LIN {X 0,Y 460.459,Z 388.647,A -85,B 0,C 180,E1 -8093.427,E2 -8093.427} C_VEL
LIN {X 0,Y 460.171,Z 393.017,A -85,B 0,C 180,E1 -8094.742,E2 -8094.742} C_VEL
LIN {X 0,Y 460.177,Z 395.283,A -85,B 0,C 180,E1 -8095.621,E2 -8095.621} C_VEL
LIN {X 0,Y 459.997,Z 397.136,A -85,B 0,C 180,E1 -8096.496,E2 -8096.496} C_VEL
LIN {X 0,Y 459.827,Z 398.543,A -85,B 0,C 180,E1 -8097.372,E2 -8097.372} C_VEL
LIN {X 0,Y 459.708,Z 400.055,A -85,B 0,C 180,E1 -8099.124,E2 -8099.124} C_VEL
LIN {X 0,Y 459.693,Z 400.219,A -85,B 0,C 180,E1 -8100,E2 -8100} C_VEL
LIN {X 0,Y 459.693,Z 399.948,A -85,B 0,C 180,E1 -8100.876,E2 -8100.876} C_VEL
LIN {X 0,Y 459.808,Z 398.188,A -85,B 0,C 180,E1 -8102.628,E2 -8102.628} C_VEL
LIN {X 0,Y 459.991,Z 396.689,A -85,B 0,C 180,E1 -8103.504,E2 -8103.504} C_VEL
LIN {X 0,Y 460.089,Z 393.615,A -85,B 0,C 180,E1 -8104.819,E2 -8104.819} C_VEL
LIN {X 0,Y 460.187,Z 388.427,A -85,B 0,C 180,E1 -8106.417,E2 -8106.417} C_VEL
LIN {X 0,Y 460.472,Z 382.079,A -85,B 0,C 180,E1 -8107.895,E2 -8107.895} C_VEL
LIN {X 0,Y 460.797,Z 374.875,A -85,B 0,C 180,E1 -8109.215,E2 -8109.215} C_VEL
LIN {X 0,Y 461.181,Z 365.885,A -85,B 0,C 180,E1 -8110.537,E2 -8110.537} C_VEL
LIN {X 0,Y 461.678,Z 356.667,A -85,B 0,C 180,E1 -8111.637,E2 -8111.637} C_VEL
LIN {X 0,Y 462.105,Z 346.45,A -85,B 0,C 180,E1 -8112.628,E2 -8112.628} C_VEL
LIN {X 0,Y 462.457,Z 334.22,A -85,B 0,C 180,E1 -8113.58,E2 -8113.58} C_VEL
LIN {X 0,Y 462.892,Z 322.561,A -85,B 0,C 180,E1 -8114.284,E2 -8114.284} C_VEL
LIN {X 0,Y 463.049,Z 309.71,A -85,B 0,C 180,E1 -8114.868,E2 -8114.868} C_VEL
LIN {X 0,Y 459.93,Z 296.427,A -85,B 0,C 180,E1 -8115.404,E2 -8115.404} C_VEL
LIN {X 0,Y 459.882,Z 292.523,A -85,B 0,C 180,E1 -8118.719,E2 -8118.719} C_VEL
LIN {X 0,Y 460.011,Z 292.186,A -85,B 0,C 180,E1 -8120.573,E2 -8120.573} C_VEL
LIN {X 0,Y 460.393,Z 292.14,A -85,B 0,C 180,E1 -8123.664,E2 -8123.664} C_VEL
LIN {X 0,Y 460.54,Z 292.115,A -85,B 0,C 180,E1 -8126.267,E2 -8126.267} C_VEL
LIN {X 0,Y 460.542,Z 292.115,A -85,B 0,C 180,E1 -8129.231,E2 -8129.231} C_VEL
LIN {X 0,Y 460.534,Z 292.118,A -85,B 0,C 180,E1 -8132.284,E2 -8132.284} C_VEL
LIN {X 0,Y 460.513,Z 292.115,A -85,B 0,C 180,E1 -8135.446,E2 -8135.446} C_VEL
LIN {X 0,Y 460.547,Z 292.114,A -85,B 0,C 180,E1 -8138.898,E2 -8138.898} C_VEL
LIN {X 0,Y 460.526,Z 292.123,A -85,B 0,C 180,E1 -8142.181,E2 -8142.181} C_VEL
LIN {X 0,Y 460.52,Z 292.119,A -85,B 0,C 180,E1 -8145.412,E2 -8145.412} C_VEL
LIN {X 0,Y 460.535,Z 292.117,A -85,B 0,C 180,E1 -8148.398,E2 -8148.398} C_VEL
LIN {X 0,Y 460.529,Z 292.12,A -85,B 0,C 180,E1 -8151.267,E2 -8151.267} C_VEL
LIN {X 0,Y 460.47,Z 292.127,A -85,B 0,C 180,E1 -8154.551,E2 -8154.551} C_VEL
LIN {X 0,Y 460.258,Z 292.271,A -85,B 0,C 180,E1 -8156.723,E2 -8156.723} C_VEL
LIN {X 0,Y 460.072,Z 297.348,A -85,B 0,C 180,E1 -8159.728,E2 -8159.728} C_VEL
LIN {X 0,Y 460.018,Z 302.263,A -85,B 0,C 180,E1 -8162.72,E2 -8162.72} C_VEL
LIN {X 0,Y 459.986,Z 307.025,A -85,B 0,C 180,E1 -8165.636,E2 -8165.636} C_VEL
LIN {X 0,Y 459.934,Z 312.249,A -85,B 0,C 180,E1 -8168.767,E2 -8168.767} C_VEL
LIN {X 0,Y 459.91,Z 316.705,A -85,B 0,C 180,E1 -8171.342,E2 -8171.342} C_VEL
LIN {X 0,Y 459.853,Z 320.715,A -85,B 0,C 180,E1 -8173.53,E2 -8173.53} C_VEL
LIN {X 0,Y 459.768,Z 322.003,A -85,B 0,C 180,E1 -8173.864,E2 -8173.864} C_VEL
LIN {X 0,Y 459.446,Z 324.926,A -85,B 0,C 180,E1 -8174.21,E2 -8174.21} C_VEL
LIN {X 0,Y 458.82,Z 329.649,A -85,B 0,C 180,E1 -8174.511,E2 -8174.511} C_VEL
LIN {X 0,Y 458.222,Z 333.723,A -85,B 0,C 180,E1 -8174.684,E2 -8174.684} C_VEL
LIN {X 0,Y 456.634,Z 345.505,A -85,B 0,C 180,E1 -8175.091,E2 -8175.091} C_VEL
LIN {X 0,Y 456.445,Z 349.068,A -85,B 0,C 180,E1 -8175.266,E2 -8175.266} C_VEL
LIN {X 0,Y 455.948,Z 360.679,A -85,B 0,C 180,E1 -8175.94,E2 -8175.94} C_VEL
LIN {X 0,Y 455.497,Z 371.287,A -85,B 0,C 180,E1 -8176.732,E2 -8176.732} C_VEL
LIN {X 0,Y 454.998,Z 382.032,A -85,B 0,C 180,E1 -8177.738,E2 -8177.738} C_VEL
LIN {X 0,Y 454.451,Z 391.614,A -85,B 0,C 180,E1 -8178.854,E2 -8178.854} C_VEL
LIN {X 0,Y 453.896,Z 400.92,A -85,B 0,C 180,E1 -8180.193,E2 -8180.193} C_VEL
LIN {X 0,Y 453.463,Z 408.307,A -85,B 0,C 180,E1 -8181.533,E2 -8181.533} C_VEL
LIN {X 0,Y 453.083,Z 415.107,A -85,B 0,C 180,E1 -8183.093,E2 -8183.093} C_VEL
LIN {X 0,Y 452.857,Z 418.931,A -85,B 0,C 180,E1 -8184.21,E2 -8184.21} C_VEL
LIN {X 0,Y 452.825,Z 422.513,A -85,B 0,C 180,E1 -8185.549,E2 -8185.549} C_VEL
LIN {X 0,Y 452.731,Z 424.363,A -85,B 0,C 180,E1 -8186.44,E2 -8186.44} C_VEL
LIN {X 0,Y 452.673,Z 425.775,A -85,B 0,C 180,E1 -8187.33,E2 -8187.33} C_VEL
LIN {X 0,Y 452.496,Z 427.385,A -85,B 0,C 180,E1 -8189.11,E2 -8189.11} C_VEL
LIN {X 0,Y 452.477,Z 427.621,A -85,B 0,C 180,E1 -8190,E2 -8190} C_VEL
LIN {X 0,Y 452.581,Z 426.849,A -85,B 0,C 180,E1 -8191.78,E2 -8191.78} C_VEL
LIN {X 0,Y 452.673,Z 425.886,A -85,B 0,C 180,E1 -8192.67,E2 -8192.67} C_VEL
LIN {X 0,Y 452.729,Z 424.535,A -85,B 0,C 180,E1 -8193.56,E2 -8193.56} C_VEL
LIN {X 0,Y 452.765,Z 421.693,A -85,B 0,C 180,E1 -8194.898,E2 -8194.898} C_VEL
LIN {X 0,Y 453.005,Z 417.822,A -85,B 0,C 180,E1 -8196.235,E2 -8196.235} C_VEL
LIN {X 0,Y 453.212,Z 412.816,A -85,B 0,C 180,E1 -8197.574,E2 -8197.574} C_VEL
LIN {X 0,Y 453.552,Z 406.493,A -85,B 0,C 180,E1 -8198.914,E2 -8198.914} C_VEL
LIN {X 0,Y 453.999,Z 398.632,A -85,B 0,C 180,E1 -8200.255,E2 -8200.255} C_VEL
LIN {X 0,Y 454.539,Z 390.597,A -85,B 0,C 180,E1 -8201.37,E2 -8201.37} C_VEL
LIN {X 0,Y 455.041,Z 380.753,A -85,B 0,C 180,E1 -8202.488,E2 -8202.488} C_VEL
LIN {X 0,Y 455.56,Z 369.521,A -85,B 0,C 180,E1 -8203.505,E2 -8203.505} C_VEL
LIN {X 0,Y 456.064,Z 358.809,A -85,B 0,C 180,E1 -8204.274,E2 -8204.274} C_VEL
LIN {X 0,Y 456.506,Z 346.692,A -85,B 0,C 180,E1 -8204.944,E2 -8204.944} C_VEL
LIN {X 0,Y 456.499,Z 339.201,A -85,B 0,C 180,E1 -8205.272,E2 -8205.272} C_VEL
LIN {X 0,Y 453.913,Z 327.065,A -85,B 0,C 180,E1 -8205.763,E2 -8205.763} C_VEL
LIN {X 0,Y 452.874,Z 322.749,A -85,B 0,C 180,E1 -8205.923,E2 -8205.923} C_VEL
LIN {X 0,Y 452.824,Z 317.039,A -85,B 0,C 180,E1 -8209.022,E2 -8209.022} C_VEL
LIN {X 0,Y 452.888,Z 312.118,A -85,B 0,C 180,E1 -8211.866,E2 -8211.866} C_VEL
LIN {X 0,Y 452.934,Z 307.318,A -85,B 0,C 180,E1 -8214.768,E2 -8214.768} C_VEL
LIN {X 0,Y 452.967,Z 302.337,A -85,B 0,C 180,E1 -8217.824,E2 -8217.824} C_VEL
LIN {X 0,Y 453.025,Z 297.475,A -85,B 0,C 180,E1 -8220.794,E2 -8220.794} C_VEL
LIN {X 0,Y 453.233,Z 293.034,A -85,B 0,C 180,E1 -8223.49,E2 -8223.49} C_VEL
LIN {X 0,Y 453.443,Z 293.004,A -85,B 0,C 180,E1 -8226.297,E2 -8226.297} C_VEL
LIN {X 0,Y 453.492,Z 292.998,A -85,B 0,C 180,E1 -8229.45,E2 -8229.45} C_VEL
LIN {X 0,Y 453.479,Z 292.999,A -85,B 0,C 180,E1 -8231.935,E2 -8231.935} C_VEL
LIN {X 0,Y 453.486,Z 292.998,A -85,B 0,C 180,E1 -8235.471,E2 -8235.471} C_VEL
LIN {X 0,Y 453.482,Z 292.997,A -85,B 0,C 180,E1 -8238.209,E2 -8238.209} C_VEL
LIN {X 0,Y 453.518,Z 292.993,A -85,B 0,C 180,E1 -8240.79,E2 -8240.79} C_VEL
LIN {X 0,Y 453.42,Z 293.008,A -85,B 0,C 180,E1 -8243.914,E2 -8243.914} C_VEL
LIN {X 0,Y 453.295,Z 293.022,A -85,B 0,C 180,E1 -8246.072,E2 -8246.072} C_VEL
LIN {X 0,Y 453.177,Z 293.167,A -85,B 0,C 180,E1 -8246.951,E2 -8246.951} C_VEL
LIN {X 0,Y 453.012,Z 298.953,A -85,B 0,C 180,E1 -8250.318,E2 -8250.318} C_VEL
LIN {X 0,Y 452.951,Z 303.959,A -85,B 0,C 180,E1 -8253.258,E2 -8253.258} C_VEL
LIN {X 0,Y 452.915,Z 309.103,A -85,B 0,C 180,E1 -8256.28,E2 -8256.28} C_VEL
LIN {X 0,Y 452.914,Z 313.849,A -85,B 0,C 180,E1 -8259.09,E2 -8259.09} C_VEL
LIN {X 0,Y 452.832,Z 318.65,A -85,B 0,C 180,E1 -8261.916,E2 -8261.916} C_VEL
LIN {X 0,Y 452.875,Z 323.053,A -85,B 0,C 180,E1 -8264.475,E2 -8264.475} C_VEL
LIN {X 0,Y 455.889,Z 337.844,A -85,B 0,C 180,E1 -8265.05,E2 -8265.05} C_VEL
LIN {X 0,Y 455.849,Z 347.577,A -85,B 0,C 180,E1 -8265.491,E2 -8265.491} C_VEL
LIN {X 0,Y 455.436,Z 359.276,A -85,B 0,C 180,E1 -8266.161,E2 -8266.161} C_VEL
LIN {X 0,Y 455.002,Z 370.542,A -85,B 0,C 180,E1 -8266.991,E2 -8266.991} C_VEL
LIN {X 0,Y 454.521,Z 382.133,A -85,B 0,C 180,E1 -8268.064,E2 -8268.064} C_VEL
LIN {X 0,Y 454.085,Z 390.947,A -85,B 0,C 180,E1 -8269.071,E2 -8269.071} C_VEL
LIN {X 0,Y 453.672,Z 400.48,A -85,B 0,C 180,E1 -8270.414,E2 -8270.414} C_VEL
LIN {X 0,Y 453.285,Z 408.148,A -85,B 0,C 180,E1 -8271.754,E2 -8271.754} C_VEL
LIN {X 0,Y 452.959,Z 414.779,A -85,B 0,C 180,E1 -8273.223,E2 -8273.223} C_VEL
LIN {X 0,Y 452.726,Z 419.813,A -85,B 0,C 180,E1 -8274.656,E2 -8274.656} C_VEL
LIN {X 0,Y 452.807,Z 422.253,A -85,B 0,C 180,E1 -8275.549,E2 -8275.549} C_VEL
LIN {X 0,Y 452.729,Z 424.241,A -85,B 0,C 180,E1 -8276.44,E2 -8276.44} C_VEL
LIN {X 0,Y 452.673,Z 425.816,A -85,B 0,C 180,E1 -8277.33,E2 -8277.33} C_VEL
LIN {X 0,Y 452.581,Z 426.923,A -85,B 0,C 180,E1 -8278.22,E2 -8278.22} C_VEL
LIN {X 0,Y 452.48,Z 427.94,A -85,B 0,C 180,E1 -8280,E2 -8280} C_VEL
LIN {X 0,Y 452.499,Z 427.804,A -85,B 0,C 180,E1 -8280.89,E2 -8280.89} C_VEL
LIN {X 0,Y 452.723,Z 426.303,A -85,B 0,C 180,E1 -8282.669,E2 -8282.669} C_VEL
LIN {X 0,Y 452.746,Z 424.917,A -85,B 0,C 180,E1 -8283.56,E2 -8283.56} C_VEL
LIN {X 0,Y 452.809,Z 422.005,A -85,B 0,C 180,E1 -8284.897,E2 -8284.897} C_VEL
LIN {X 0,Y 453,Z 418.002,A -85,B 0,C 180,E1 -8286.235,E2 -8286.235} C_VEL
LIN {X 0,Y 453.266,Z 411.852,A -85,B 0,C 180,E1 -8287.797,E2 -8287.797} C_VEL
LIN {X 0,Y 453.627,Z 405.037,A -85,B 0,C 180,E1 -8289.137,E2 -8289.137} C_VEL
LIN {X 0,Y 454.045,Z 396.508,A -85,B 0,C 180,E1 -8290.479,E2 -8290.479} C_VEL
LIN {X 0,Y 454.517,Z 386.739,A -85,B 0,C 180,E1 -8291.709,E2 -8291.709} C_VEL
LIN {X 0,Y 455.048,Z 376.108,A -85,B 0,C 180,E1 -8292.785,E2 -8292.785} C_VEL
LIN {X 0,Y 455.43,Z 365.151,A -85,B 0,C 180,E1 -8293.674,E2 -8293.674} C_VEL
LIN {X 0,Y 455.951,Z 351.977,A -85,B 0,C 180,E1 -8294.506,E2 -8294.506} C_VEL
LIN {X 0,Y 456.235,Z 338.735,A -85,B 0,C 180,E1 -8295.124,E2 -8295.124} C_VEL
LIN {X 0,Y 453.546,Z 327.053,A -85,B 0,C 180,E1 -8295.627,E2 -8295.627} C_VEL
LIN {X 0,Y 453.092,Z 325.142,A -85,B 0,C 180,E1 -8295.719,E2 -8295.719} C_VEL
LIN {X 0,Y 453.099,Z 319.349,A -85,B 0,C 180,E1 -8299.01,E2 -8299.01} C_VEL
LIN {X 0,Y 453.102,Z 314.205,A -85,B 0,C 180,E1 -8301.855,E2 -8301.855} C_VEL
LIN {X 0,Y 453.091,Z 308.727,A -85,B 0,C 180,E1 -8304.759,E2 -8304.759} C_VEL
LIN {X 0,Y 453.096,Z 302.547,A -85,B 0,C 180,E1 -8307.855,E2 -8307.855} C_VEL
LIN {X 0,Y 453.124,Z 297.403,A -85,B 0,C 180,E1 -8310.27,E2 -8310.27} C_VEL
LIN {X 0,Y 453.155,Z 293.042,A -85,B 0,C 180,E1 -8312.282,E2 -8312.282} C_VEL
LIN {X 0,Y 453.426,Z 293.008,A -85,B 0,C 180,E1 -8314.994,E2 -8314.994} C_VEL
LIN {X 0,Y 453.465,Z 293.001,A -85,B 0,C 180,E1 -8318.312,E2 -8318.312} C_VEL
LIN {X 0,Y 453.495,Z 292.997,A -85,B 0,C 180,E1 -8320.609,E2 -8320.609} C_VEL
LIN {X 0,Y 453.465,Z 293.001,A -85,B 0,C 180,E1 -8324.221,E2 -8324.221} C_VEL
LIN {X 0,Y 453.451,Z 293.002,A -85,B 0,C 180,E1 -8327.003,E2 -8327.003} C_VEL
LIN {X 0,Y 453.497,Z 293.118,A -85,B 0,C 180,E1 -8327.722,E2 -8327.722} C_VEL
LIN {X 0,Y 455.009,Z 300.676,A -85,B 0,C 180,E1 -8330.707,E2 -8330.707} C_VEL
LIN {X 0,Y 456.188,Z 307.36,A -85,B 0,C 180,E1 -8333.236,E2 -8333.236} C_VEL
LIN {X 0,Y 456.148,Z 311.66,A -85,B 0,C 180,E1 -8334.745,E2 -8334.745} C_VEL
LIN {X 0,Y 455.594,Z 320.505,A -85,B 0,C 180,E1 -8337.743,E2 -8337.743} C_VEL
LIN {X 0,Y 455.028,Z 330.087,A -85,B 0,C 180,E1 -8340.887,E2 -8340.887} C_VEL
LIN {X 0,Y 454.434,Z 340.853,A -85,B 0,C 180,E1 -8344.34,E2 -8344.34} C_VEL
LIN {X 0,Y 454.121,Z 348.746,A -85,B 0,C 180,E1 -8346.756,E2 -8346.756} C_VEL
LIN {X 0,Y 453.704,Z 359.926,A -85,B 0,C 180,E1 -8350.075,E2 -8350.075} C_VEL
LIN {X 0,Y 453.322,Z 370.951,A -85,B 0,C 180,E1 -8353.333,E2 -8353.333} C_VEL
LIN {X 0,Y 453.268,Z 373.395,A -85,B 0,C 180,E1 -8354.067,E2 -8354.067} C_VEL
LIN {X 0,Y 455.379,Z 386.776,A -85,B 0,C 180,E1 -8354.499,E2 -8354.499} C_VEL
LIN {X 0,Y 456.369,Z 394.506,A -85,B 0,C 180,E1 -8354.823,E2 -8354.823} C_VEL
LIN {X 0,Y 455.942,Z 406.083,A -85,B 0,C 180,E1 -8355.38,E2 -8355.38} C_VEL
LIN {X 0,Y 455.318,Z 418.38,A -85,B 0,C 180,E1 -8356.158,E2 -8356.158} C_VEL
LIN {X 0,Y 454.807,Z 429.198,A -85,B 0,C 180,E1 -8357.033,E2 -8357.033} C_VEL
LIN {X 0,Y 454.406,Z 438.408,A -85,B 0,C 180,E1 -8357.948,E2 -8357.948} C_VEL
LIN {X 0,Y 453.8,Z 447.655,A -85,B 0,C 180,E1 -8359.064,E2 -8359.064} C_VEL
LIN {X 0,Y 453.346,Z 456.683,A -85,B 0,C 180,E1 -8360.407,E2 -8360.407} C_VEL
LIN {X 0,Y 452.999,Z 463.957,A -85,B 0,C 180,E1 -8361.749,E2 -8361.749} C_VEL
LIN {X 0,Y 452.762,Z 468.874,A -85,B 0,C 180,E1 -8362.867,E2 -8362.867} C_VEL
LIN {X 0,Y 452.678,Z 473.664,A -85,B 0,C 180,E1 -8364.208,E2 -8364.208} C_VEL
LIN {X 0,Y 452.501,Z 477.314,A -85,B 0,C 180,E1 -8365.546,E2 -8365.546} C_VEL
LIN {X 0,Y 452.513,Z 479.204,A -85,B 0,C 180,E1 -8366.438,E2 -8366.438} C_VEL
LIN {X 0,Y 452.496,Z 480.621,A -85,B 0,C 180,E1 -8367.329,E2 -8367.329} C_VEL
LIN {X 0,Y 452.463,Z 481.628,A -85,B 0,C 180,E1 -8368.22,E2 -8368.22} C_VEL
LIN {X 0,Y 452.433,Z 482.241,A -85,B 0,C 180,E1 -8369.11,E2 -8369.11} C_VEL
LIN {X 0,Y 452.41,Z 482.453,A -85,B 0,C 180,E1 -8370,E2 -8370} C_VEL
LIN {X 0,Y 452.433,Z 482.232,A -85,B 0,C 180,E1 -8370.89,E2 -8370.89} C_VEL
LIN {X 0,Y 452.463,Z 481.613,A -85,B 0,C 180,E1 -8371.78,E2 -8371.78} C_VEL
LIN {X 0,Y 452.496,Z 480.598,A -85,B 0,C 180,E1 -8372.671,E2 -8372.671} C_VEL
LIN {X 0,Y 452.513,Z 479.167,A -85,B 0,C 180,E1 -8373.562,E2 -8373.562} C_VEL
LIN {X 0,Y 452.567,Z 476.17,A -85,B 0,C 180,E1 -8374.9,E2 -8374.9} C_VEL
LIN {X 0,Y 452.691,Z 471.23,A -85,B 0,C 180,E1 -8376.486,E2 -8376.486} C_VEL
LIN {X 0,Y 452.926,Z 464.854,A -85,B 0,C 180,E1 -8378.028,E2 -8378.028} C_VEL
LIN {X 0,Y 453.299,Z 457.819,A -85,B 0,C 180,E1 -8379.369,E2 -8379.369} C_VEL
LIN {X 0,Y 453.708,Z 449.019,A -85,B 0,C 180,E1 -8380.713,E2 -8380.713} C_VEL
LIN {X 0,Y 454.27,Z 440.028,A -85,B 0,C 180,E1 -8381.829,E2 -8381.829} C_VEL
LIN {X 0,Y 454.755,Z 430.118,A -85,B 0,C 180,E1 -8382.84,E2 -8382.84} C_VEL
LIN {X 0,Y 455.196,Z 419.398,A -85,B 0,C 180,E1 -8383.732,E2 -8383.732} C_VEL
LIN {X 0,Y 455.743,Z 407.42,A -85,B 0,C 180,E1 -8384.513,E2 -8384.513} C_VEL
LIN {X 0,Y 456.296,Z 395.104,A -85,B 0,C 180,E1 -8385.122,E2 -8385.122} C_VEL
LIN {X 0,Y 455.375,Z 386.762,A -85,B 0,C 180,E1 -8385.478,E2 -8385.478} C_VEL
LIN {X 0,Y 453.435,Z 374.456,A -85,B 0,C 180,E1 -8385.885,E2 -8385.885} C_VEL
LIN {X 0,Y 453.219,Z 372.318,A -85,B 0,C 180,E1 -8385.965,E2 -8385.965} C_VEL
LIN {X 0,Y 453.519,Z 361.56,A -85,B 0,C 180,E1 -8389.039,E2 -8389.039} C_VEL
LIN {X 0,Y 453.874,Z 350.262,A -85,B 0,C 180,E1 -8392.295,E2 -8392.295} C_VEL
LIN {X 0,Y 454.267,Z 338.832,A -85,B 0,C 180,E1 -8395.67,E2 -8395.67} C_VEL
LIN {X 0,Y 454.725,Z 327.585,A -85,B 0,C 180,E1 -8399.134,E2 -8399.134} C_VEL
LIN {X 0,Y 455.109,Z 319.203,A -85,B 0,C 180,E1 -8401.86,E2 -8401.86} C_VEL
LIN {X 0,Y 455.763,Z 309.699,A -85,B 0,C 180,E1 -8405.187,E2 -8405.187} C_VEL
LIN {X 0,Y 455.798,Z 305.785,A -85,B 0,C 180,E1 -8406.698,E2 -8406.698} C_VEL
LIN {X 0,Y 454.8,Z 299.736,A -85,B 0,C 180,E1 -8409.408,E2 -8409.408} C_VEL
LIN {X 0,Y 453.857,Z 295.018,A -85,B 0,C 180,E1 -8411.988,E2 -8411.988} C_VEL
LIN {X 0,Y 453.459,Z 293.004,A -85,B 0,C 180,E1 -8413.431,E2 -8413.431} C_VEL
LIN {X 0,Y 453.462,Z 293.003,A -85,B 0,C 180,E1 -8415.778,E2 -8415.778} C_VEL
LIN {X 0,Y 453.496,Z 292.997,A -85,B 0,C 180,E1 -8419.409,E2 -8419.409} C_VEL
LIN {X 0,Y 453.451,Z 293.004,A -85,B 0,C 180,E1 -8422.227,E2 -8422.227} C_VEL
LIN {X 0,Y 453.49,Z 292.997,A -85,B 0,C 180,E1 -8425.223,E2 -8425.223} C_VEL
LIN {X 0,Y 453.469,Z 293.001,A -85,B 0,C 180,E1 -8428.475,E2 -8428.475} C_VEL
LIN {X 0,Y 453.532,Z 292.995,A -85,B 0,C 180,E1 -8432.041,E2 -8432.041} C_VEL
LIN {X 0,Y 453.532,Z 293.311,A -85,B 0,C 180,E1 -8434.285,E2 -8434.285} C_VEL
LIN {X 0,Y 453.636,Z 294.763,A -85,B 0,C 180,E1 -8436.246,E2 -8436.246} C_VEL
LIN {X 0,Y 453.555,Z 297.019,A -85,B 0,C 180,E1 -8439.121,E2 -8439.121} C_VEL
LIN {X 0,Y 453.459,Z 299.324,A -85,B 0,C 180,E1 -8441.942,E2 -8441.942} C_VEL
LIN {X 0,Y 453.454,Z 301.623,A -85,B 0,C 180,E1 -8444.425,E2 -8444.425} C_VEL
LIN {X 0,Y 456.607,Z 312.569,A -85,B 0,C 180,E1 -8444.931,E2 -8444.931} C_VEL
LIN {X 0,Y 456.284,Z 325.957,A -85,B 0,C 180,E1 -8445.562,E2 -8445.562} C_VEL
LIN {X 0,Y 455.928,Z 337.302,A -85,B 0,C 180,E1 -8446.275,E2 -8446.275} C_VEL
LIN {X 0,Y 455.474,Z 348.667,A -85,B 0,C 180,E1 -8447.185,E2 -8447.185} C_VEL
LIN {X 0,Y 454.99,Z 358.83,A -85,B 0,C 180,E1 -8448.19,E2 -8448.19} C_VEL
LIN {X 0,Y 454.517,Z 367.958,A -85,B 0,C 180,E1 -8449.307,E2 -8449.307} C_VEL
LIN {X 0,Y 454.079,Z 376.775,A -85,B 0,C 180,E1 -8450.647,E2 -8450.647} C_VEL
LIN {X 0,Y 453.692,Z 383.842,A -85,B 0,C 180,E1 -8451.986,E2 -8451.986} C_VEL
LIN {X 0,Y 453.452,Z 389.413,A -85,B 0,C 180,E1 -8453.325,E2 -8453.325} C_VEL
LIN {X 0,Y 453.15,Z 393.765,A -85,B 0,C 180,E1 -8454.661,E2 -8454.661} C_VEL
LIN {X 0,Y 453.15,Z 396.02,A -85,B 0,C 180,E1 -8455.552,E2 -8455.552} C_VEL
LIN {X 0,Y 452.959,Z 397.869,A -85,B 0,C 180,E1 -8456.442,E2 -8456.442} C_VEL
LIN {X 0,Y 452.776,Z 399.268,A -85,B 0,C 180,E1 -8457.331,E2 -8457.331} C_VEL
LIN {X 0,Y 452.683,Z 400.214,A -85,B 0,C 180,E1 -8458.221,E2 -8458.221} C_VEL
LIN {X 0,Y 452.644,Z 400.761,A -85,B 0,C 180,E1 -8459.11,E2 -8459.11} C_VEL
LIN {X 0,Y 452.628,Z 400.914,A -85,B 0,C 180,E1 -8460,E2 -8460} C_VEL
LIN {X 0,Y 452.627,Z 400.626,A -85,B 0,C 180,E1 -8460.89,E2 -8460.89} C_VEL
LIN {X 0,Y 452.649,Z 399.929,A -85,B 0,C 180,E1 -8461.78,E2 -8461.78} C_VEL
LIN {X 0,Y 452.759,Z 398.828,A -85,B 0,C 180,E1 -8462.669,E2 -8462.669} C_VEL
LIN {X 0,Y 452.952,Z 397.306,A -85,B 0,C 180,E1 -8463.558,E2 -8463.558} C_VEL
LIN {X 0,Y 453.044,Z 394.197,A -85,B 0,C 180,E1 -8464.895,E2 -8464.895} C_VEL
LIN {X 0,Y 453.076,Z 390.021,A -85,B 0,C 180,E1 -8466.234,E2 -8466.234} C_VEL
LIN {X 0,Y 453.422,Z 383.597,A -85,B 0,C 180,E1 -8467.795,E2 -8467.795} C_VEL
LIN {X 0,Y 453.733,Z 376.611,A -85,B 0,C 180,E1 -8469.135,E2 -8469.135} C_VEL
LIN {X 0,Y 454.047,Z 369.485,A -85,B 0,C 180,E1 -8470.254,E2 -8470.254} C_VEL
LIN {X 0,Y 454.497,Z 360.887,A -85,B 0,C 180,E1 -8471.371,E2 -8471.371} C_VEL
LIN {X 0,Y 454.959,Z 350.28,A -85,B 0,C 180,E1 -8472.49,E2 -8472.49} C_VEL
LIN {X 0,Y 455.447,Z 338.649,A -85,B 0,C 180,E1 -8473.475,E2 -8473.475} C_VEL
LIN {X 0,Y 455.822,Z 326.434,A -85,B 0,C 180,E1 -8474.282,E2 -8474.282} C_VEL
LIN {X 0,Y 456.254,Z 312.971,A -85,B 0,C 180,E1 -8474.952,E2 -8474.952} C_VEL
LIN {X 0,Y 455.938,Z 310.072,A -85,B 0,C 180,E1 -8475.077,E2 -8475.077} C_VEL
LIN {X 0,Y 452.862,Z 296.968,A -85,B 0,C 180,E1 -8475.615,E2 -8475.615} C_VEL
LIN {X 0,Y 452.819,Z 293.084,A -85,B 0,C 180,E1 -8479.022,E2 -8479.022} C_VEL
LIN {X 0,Y 453.13,Z 293.041,A -85,B 0,C 180,E1 -8481.854,E2 -8481.854} C_VEL
LIN {X 0,Y 453.419,Z 293.007,A -85,B 0,C 180,E1 -8484.74,E2 -8484.74} C_VEL
LIN {X 0,Y 453.532,Z 292.987,A -85,B 0,C 180,E1 -8487.959,E2 -8487.959} C_VEL
LIN {X 0,Y 453.468,Z 292.992,A -85,B 0,C 180,E1 -8491.525,E2 -8491.525} C_VEL
LIN {X 0,Y 453.49,Z 292.992,A -85,B 0,C 180,E1 -8494.777,E2 -8494.777} C_VEL
LIN {X 0,Y 453.467,Z 293.001,A -85,B 0,C 180,E1 -8498.312,E2 -8498.312} C_VEL
LIN {X 0,Y 453.497,Z 292.996,A -85,B 0,C 180,E1 -8500.609,E2 -8500.609} C_VEL
LIN {X 0,Y 453.459,Z 292.999,A -85,B 0,C 180,E1 -8503.244,E2 -8503.244} C_VEL
LIN {X 0,Y 453.469,Z 293.002,A -85,B 0,C 180,E1 -8505.779,E2 -8505.779} C_VEL
LIN {X 0,Y 453.482,Z 292.997,A -85,B 0,C 180,E1 -8508.209,E2 -8508.209} C_VEL
LIN {X 0,Y 453.497,Z 292.993,A -85,B 0,C 180,E1 -8510.793,E2 -8510.793} C_VEL
LIN {X 0,Y 453.442,Z 293.006,A -85,B 0,C 180,E1 -8513.916,E2 -8513.916} C_VEL
LIN {X 0,Y 453.224,Z 293.13,A -85,B 0,C 180,E1 -8516.729,E2 -8516.729} C_VEL
LIN {X 0,Y 453.006,Z 299.125,A -85,B 0,C 180,E1 -8520.319,E2 -8520.319} C_VEL
LIN {X 0,Y 452.966,Z 303.944,A -85,B 0,C 180,E1 -8523.259,E2 -8523.259} C_VEL
LIN {X 0,Y 452.913,Z 308.879,A -85,B 0,C 180,E1 -8526.281,E2 -8526.281} C_VEL
LIN {X 0,Y 452.873,Z 313.58,A -85,B 0,C 180,E1 -8529.088,E2 -8529.088} C_VEL
LIN {X 0,Y 452.821,Z 318.552,A -85,B 0,C 180,E1 -8531.916,E2 -8531.916} C_VEL
LIN {X 0,Y 452.857,Z 322.861,A -85,B 0,C 180,E1 -8534.196,E2 -8534.196} C_VEL
LIN {X 0,Y 455.916,Z 336.043,A -85,B 0,C 180,E1 -8534.679,E2 -8534.679} C_VEL
LIN {X 0,Y 456.622,Z 340.8,A -85,B 0,C 180,E1 -8534.889,E2 -8534.889} C_VEL
LIN {X 0,Y 456.445,Z 349.068,A -85,B 0,C 180,E1 -8535.266,E2 -8535.266} C_VEL
LIN {X 0,Y 455.71,Z 354.62,A -85,B 0,C 180,E1 -8535.546,E2 -8535.546} C_VEL
LIN {X 0,Y 452.572,Z 363.35,A -85,B 0,C 180,E1 -8536.003,E2 -8536.003} C_VEL
LIN {X 0,Y 449.32,Z 371.611,A -85,B 0,C 180,E1 -8536.542,E2 -8536.542} C_VEL
LIN {X 0,Y 448.395,Z 376.399,A -85,B 0,C 180,E1 -8536.944,E2 -8536.944} C_VEL
LIN {X 0,Y 447.864,Z 386.531,A -85,B 0,C 180,E1 -8537.999,E2 -8537.999} C_VEL
LIN {X 0,Y 447.275,Z 395.361,A -85,B 0,C 180,E1 -8539.131,E2 -8539.131} C_VEL
LIN {X 0,Y 446.778,Z 403.968,A -85,B 0,C 180,E1 -8540.493,E2 -8540.493} C_VEL
LIN {X 0,Y 446.322,Z 410.872,A -85,B 0,C 180,E1 -8541.853,E2 -8541.853} C_VEL
LIN {X 0,Y 446.042,Z 416.864,A -85,B 0,C 180,E1 -8543.361,E2 -8543.361} C_VEL
LIN {X 0,Y 445.728,Z 421.872,A -85,B 0,C 180,E1 -8545.025,E2 -8545.025} C_VEL
LIN {X 0,Y 445.67,Z 424.778,A -85,B 0,C 180,E1 -8546.383,E2 -8546.383} C_VEL
LIN {X 0,Y 445.594,Z 426.191,A -85,B 0,C 180,E1 -8547.288,E2 -8547.288} C_VEL
LIN {X 0,Y 445.433,Z 427.799,A -85,B 0,C 180,E1 -8549.096,E2 -8549.096} C_VEL
LIN {X 0,Y 445.412,Z 428.034,A -85,B 0,C 180,E1 -8550,E2 -8550} C_VEL
LIN {X 0,Y 445.524,Z 427.261,A -85,B 0,C 180,E1 -8551.808,E2 -8551.808} C_VEL
LIN {X 0,Y 445.594,Z 426.3,A -85,B 0,C 180,E1 -8552.712,E2 -8552.712} C_VEL
LIN {X 0,Y 445.668,Z 424.948,A -85,B 0,C 180,E1 -8553.617,E2 -8553.617} C_VEL
LIN {X 0,Y 445.683,Z 422.107,A -85,B 0,C 180,E1 -8554.976,E2 -8554.976} C_VEL
LIN {X 0,Y 446.043,Z 417.178,A -85,B 0,C 180,E1 -8556.64,E2 -8556.64} C_VEL
LIN {X 0,Y 446.287,Z 411.266,A -85,B 0,C 180,E1 -8558.148,E2 -8558.148} C_VEL
LIN {X 0,Y 446.75,Z 404.49,A -85,B 0,C 180,E1 -8559.508,E2 -8559.508} C_VEL
LIN {X 0,Y 447.24,Z 396.001,A -85,B 0,C 180,E1 -8560.869,E2 -8560.869} C_VEL
LIN {X 0,Y 447.789,Z 387.303,A -85,B 0,C 180,E1 -8562.003,E2 -8562.003} C_VEL
LIN {X 0,Y 448.331,Z 377.763,A -85,B 0,C 180,E1 -8563.022,E2 -8563.022} C_VEL
LIN {X 0,Y 448.753,Z 367.721,A -85,B 0,C 180,E1 -8563.895,E2 -8563.895} C_VEL
LIN {X 0,Y 449.376,Z 355.498,A -85,B 0,C 180,E1 -8564.723,E2 -8564.723} C_VEL
LIN {X 0,Y 449.749,Z 343.394,A -85,B 0,C 180,E1 -8565.348,E2 -8565.348} C_VEL
LIN {X 0,Y 449.409,Z 338.943,A -85,B 0,C 180,E1 -8565.545,E2 -8565.545} C_VEL
LIN {X 0,Y 446.675,Z 326.704,A -85,B 0,C 180,E1 -8566.043,E2 -8566.043} C_VEL
LIN {X 0,Y 445.823,Z 323.129,A -85,B 0,C 180,E1 -8566.168,E2 -8566.168} C_VEL
LIN {X 0,Y 445.777,Z 317.308,A -85,B 0,C 180,E1 -8569.334,E2 -8569.334} C_VEL
LIN {X 0,Y 445.838,Z 312.317,A -85,B 0,C 180,E1 -8572.23,E2 -8572.23} C_VEL
LIN {X 0,Y 445.871,Z 307.446,A -85,B 0,C 180,E1 -8575.188,E2 -8575.188} C_VEL
LIN {X 0,Y 445.915,Z 302.515,A -85,B 0,C 180,E1 -8578.218,E2 -8578.218} C_VEL
LIN {X 0,Y 446.004,Z 297.418,A -85,B 0,C 180,E1 -8581.333,E2 -8581.333} C_VEL
LIN {X 0,Y 446.196,Z 293.911,A -85,B 0,C 180,E1 -8583.455,E2 -8583.455} C_VEL
LIN {X 0,Y 446.383,Z 293.885,A -85,B 0,C 180,E1 -8585.63,E2 -8585.63} C_VEL
LIN {X 0,Y 446.446,Z 293.875,A -85,B 0,C 180,E1 -8589.027,E2 -8589.027} C_VEL
LIN {X 0,Y 446.437,Z 293.878,A -85,B 0,C 180,E1 -8592.277,E2 -8592.277} C_VEL
LIN {X 0,Y 446.454,Z 293.876,A -85,B 0,C 180,E1 -8595.104,E2 -8595.104} C_VEL
LIN {X 0,Y 446.431,Z 293.877,A -85,B 0,C 180,E1 -8598.609,E2 -8598.609} C_VEL
LIN {X 0,Y 446.462,Z 293.872,A -85,B 0,C 180,E1 -8600.975,E2 -8600.975} C_VEL
LIN {X 0,Y 446.351,Z 293.885,A -85,B 0,C 180,E1 -8604.367,E2 -8604.367} C_VEL
LIN {X 0,Y 446.114,Z 294.029,A -85,B 0,C 180,E1 -8606.977,E2 -8606.977} C_VEL
LIN {X 0,Y 445.925,Z 300.491,A -85,B 0,C 180,E1 -8610.753,E2 -8610.753} C_VEL
LIN {X 0,Y 445.89,Z 305.898,A -85,B 0,C 180,E1 -8613.952,E2 -8613.952} C_VEL
LIN {X 0,Y 445.833,Z 310.709,A -85,B 0,C 180,E1 -8616.79,E2 -8616.79} C_VEL
LIN {X 0,Y 445.802,Z 315.622,A -85,B 0,C 180,E1 -8619.707,E2 -8619.707} C_VEL
LIN {X 0,Y 445.764,Z 320.486,A -85,B 0,C 180,E1 -8622.569,E2 -8622.569} C_VEL
LIN {X 0,Y 445.798,Z 323.351,A -85,B 0,C 180,E1 -8624.26,E2 -8624.26} C_VEL
LIN {X 0,Y 448.684,Z 337.591,A -85,B 0,C 180,E1 -8624.819,E2 -8624.819} C_VEL
LIN {X 0,Y 449.16,Z 341.126,A -85,B 0,C 180,E1 -8624.98,E2 -8624.98} C_VEL
LIN {X 0,Y 448.721,Z 353.497,A -85,B 0,C 180,E1 -8625.603,E2 -8625.603} C_VEL
LIN {X 0,Y 448.224,Z 365.545,A -85,B 0,C 180,E1 -8626.397,E2 -8626.397} C_VEL
LIN {X 0,Y 447.786,Z 377.584,A -85,B 0,C 180,E1 -8627.422,E2 -8627.422} C_VEL
LIN {X 0,Y 447.293,Z 387.294,A -85,B 0,C 180,E1 -8628.444,E2 -8628.444} C_VEL
LIN {X 0,Y 446.847,Z 396.102,A -85,B 0,C 180,E1 -8629.579,E2 -8629.579} C_VEL
LIN {X 0,Y 446.415,Z 404.734,A -85,B 0,C 180,E1 -8630.942,E2 -8630.942} C_VEL
LIN {X 0,Y 446.106,Z 411.635,A -85,B 0,C 180,E1 -8632.304,E2 -8632.304} C_VEL
LIN {X 0,Y 445.925,Z 417.133,A -85,B 0,C 180,E1 -8633.666,E2 -8633.666} C_VEL
LIN {X 0,Y 445.654,Z 421.429,A -85,B 0,C 180,E1 -8635.024,E2 -8635.024} C_VEL
LIN {X 0,Y 445.667,Z 424.622,A -85,B 0,C 180,E1 -8636.383,E2 -8636.383} C_VEL
LIN {X 0,Y 445.594,Z 426.216,A -85,B 0,C 180,E1 -8637.288,E2 -8637.288} C_VEL
LIN {X 0,Y 445.524,Z 427.342,A -85,B 0,C 180,E1 -8638.192,E2 -8638.192} C_VEL
LIN {X 0,Y 445.415,Z 428.384,A -85,B 0,C 180,E1 -8640,E2 -8640} C_VEL
LIN {X 0,Y 445.437,Z 428.262,A -85,B 0,C 180,E1 -8640.904,E2 -8640.904} C_VEL
LIN {X 0,Y 445.671,Z 426.778,A -85,B 0,C 180,E1 -8642.712,E2 -8642.712} C_VEL
LIN {X 0,Y 445.684,Z 425.406,A -85,B 0,C 180,E1 -8643.616,E2 -8643.616} C_VEL
LIN {X 0,Y 445.756,Z 422.509,A -85,B 0,C 180,E1 -8644.975,E2 -8644.975} C_VEL
LIN {X 0,Y 445.97,Z 418.523,A -85,B 0,C 180,E1 -8646.333,E2 -8646.333} C_VEL
LIN {X 0,Y 446.261,Z 412.371,A -85,B 0,C 180,E1 -8647.921,E2 -8647.921} C_VEL
LIN {X 0,Y 446.654,Z 405.555,A -85,B 0,C 180,E1 -8649.281,E2 -8649.281} C_VEL
LIN {X 0,Y 447.095,Z 397.016,A -85,B 0,C 180,E1 -8650.644,E2 -8650.644} C_VEL
LIN {X 0,Y 447.588,Z 387.258,A -85,B 0,C 180,E1 -8651.893,E2 -8651.893} C_VEL
LIN {X 0,Y 448.093,Z 377.832,A -85,B 0,C 180,E1 -8652.875,E2 -8652.875} C_VEL
LIN {X 0,Y 448.522,Z 366.965,A -85,B 0,C 180,E1 -8653.802,E2 -8653.802} C_VEL
LIN {X 0,Y 449.017,Z 354.636,A -85,B 0,C 180,E1 -8654.619,E2 -8654.619} C_VEL
LIN {X 0,Y 449.49,Z 342.348,A -85,B 0,C 180,E1 -8655.241,E2 -8655.241} C_VEL
LIN {X 0,Y 449.159,Z 338.567,A -85,B 0,C 180,E1 -8655.412,E2 -8655.412} C_VEL
LIN {X 0,Y 446.449,Z 327.413,A -85,B 0,C 180,E1 -8655.907,E2 -8655.907} C_VEL
LIN {X 0,Y 446.06,Z 325.706,A -85,B 0,C 180,E1 -8655.983,E2 -8655.983} C_VEL
LIN {X 0,Y 446.065,Z 319.848,A -85,B 0,C 180,E1 -8659.321,E2 -8659.321} C_VEL
LIN {X 0,Y 446.078,Z 314.584,A -85,B 0,C 180,E1 -8662.217,E2 -8662.217} C_VEL
LIN {X 0,Y 446.062,Z 309.023,A -85,B 0,C 180,E1 -8665.176,E2 -8665.176} C_VEL
LIN {X 0,Y 446.083,Z 302.999,A -85,B 0,C 180,E1 -8668.206,E2 -8668.206} C_VEL
LIN {X 0,Y 446.161,Z 297.544,A -85,B 0,C 180,E1 -8670.794,E2 -8670.794} C_VEL
LIN {X 0,Y 446.14,Z 293.916,A -85,B 0,C 180,E1 -8672.451,E2 -8672.451} C_VEL
LIN {X 0,Y 446.379,Z 293.886,A -85,B 0,C 180,E1 -8675.043,E2 -8675.043} C_VEL
LIN {X 0,Y 446.417,Z 293.88,A -85,B 0,C 180,E1 -8678.079,E2 -8678.079} C_VEL
LIN {X 0,Y 446.424,Z 293.878,A -85,B 0,C 180,E1 -8680.917,E2 -8680.917} C_VEL
LIN {X 0,Y 446.402,Z 293.881,A -85,B 0,C 180,E1 -8683.846,E2 -8683.846} C_VEL
LIN {X 0,Y 446.433,Z 293.877,A -85,B 0,C 180,E1 -8686.78,E2 -8686.78} C_VEL
LIN {X 0,Y 446.455,Z 294.081,A -85,B 0,C 180,E1 -8687.398,E2 -8687.398} C_VEL
LIN {X 0,Y 447.896,Z 301.146,A -85,B 0,C 180,E1 -8690.252,E2 -8690.252} C_VEL
LIN {X 0,Y 449.156,Z 308.137,A -85,B 0,C 180,E1 -8692.94,E2 -8692.94} C_VEL
LIN {X 0,Y 449.25,Z 312.275,A -85,B 0,C 180,E1 -8694.438,E2 -8694.438} C_VEL
LIN {X 0,Y 448.684,Z 320.545,A -85,B 0,C 180,E1 -8697.29,E2 -8697.29} C_VEL
LIN {X 0,Y 448.101,Z 329.82,A -85,B 0,C 180,E1 -8700.393,E2 -8700.393} C_VEL
LIN {X 0,Y 447.476,Z 340.593,A -85,B 0,C 180,E1 -8703.911,E2 -8703.911} C_VEL
LIN {X 0,Y 447.136,Z 348.387,A -85,B 0,C 180,E1 -8706.371,E2 -8706.371} C_VEL
LIN {X 0,Y 446.734,Z 357.98,A -85,B 0,C 180,E1 -8709.27,E2 -8709.27} C_VEL
LIN {X 0,Y 446.315,Z 368.939,A -85,B 0,C 180,E1 -8712.591,E2 -8712.591} C_VEL
LIN {X 0,Y 446.188,Z 372.873,A -85,B 0,C 180,E1 -8713.792,E2 -8713.792} C_VEL
LIN {X 0,Y 448.476,Z 387.44,A -85,B 0,C 180,E1 -8714.293,E2 -8714.293} C_VEL
LIN {X 0,Y 449.443,Z 395.306,A -85,B 0,C 180,E1 -8714.642,E2 -8714.642} C_VEL
LIN {X 0,Y 448.957,Z 407.508,A -85,B 0,C 180,E1 -8715.263,E2 -8715.263} C_VEL
LIN {X 0,Y 448.324,Z 419.337,A -85,B 0,C 180,E1 -8716.053,E2 -8716.053} C_VEL
LIN {X 0,Y 447.755,Z 430.444,A -85,B 0,C 180,E1 -8717.002,E2 -8717.002} C_VEL
LIN {X 0,Y 447.293,Z 439.794,A -85,B 0,C 180,E1 -8717.984,E2 -8717.984} C_VEL
LIN {X 0,Y 446.685,Z 448.708,A -85,B 0,C 180,E1 -8719.117,E2 -8719.117} C_VEL
LIN {X 0,Y 446.24,Z 457.436,A -85,B 0,C 180,E1 -8720.481,E2 -8720.481} C_VEL
LIN {X 0,Y 445.884,Z 464.415,A -85,B 0,C 180,E1 -8721.845,E2 -8721.845} C_VEL
LIN {X 0,Y 445.649,Z 470.017,A -85,B 0,C 180,E1 -8723.208,E2 -8723.208} C_VEL
LIN {X 0,Y 445.562,Z 474.416,A -85,B 0,C 180,E1 -8724.569,E2 -8724.569} C_VEL
LIN {X 0,Y 445.427,Z 476.736,A -85,B 0,C 180,E1 -8725.475,E2 -8725.475} C_VEL
LIN {X 0,Y 445.422,Z 478.623,A -85,B 0,C 180,E1 -8726.381,E2 -8726.381} C_VEL
LIN {X 0,Y 445.424,Z 480.042,A -85,B 0,C 180,E1 -8727.287,E2 -8727.287} C_VEL
LIN {X 0,Y 445.411,Z 481.049,A -85,B 0,C 180,E1 -8728.192,E2 -8728.192} C_VEL
LIN {X 0,Y 445.373,Z 481.657,A -85,B 0,C 180,E1 -8729.096,E2 -8729.096} C_VEL
LIN {X 0,Y 445.349,Z 481.863,A -85,B 0,C 180,E1 -8730,E2 -8730} C_VEL
LIN {X 0,Y 445.373,Z 481.636,A -85,B 0,C 180,E1 -8730.904,E2 -8730.904} C_VEL
LIN {X 0,Y 445.411,Z 481.012,A -85,B 0,C 180,E1 -8731.808,E2 -8731.808} C_VEL
LIN {X 0,Y 445.424,Z 479.987,A -85,B 0,C 180,E1 -8732.713,E2 -8732.713} C_VEL
LIN {X 0,Y 445.438,Z 478.542,A -85,B 0,C 180,E1 -8733.618,E2 -8733.618} C_VEL
LIN {X 0,Y 445.504,Z 475.528,A -85,B 0,C 180,E1 -8734.978,E2 -8734.978} C_VEL
LIN {X 0,Y 445.627,Z 470.898,A -85,B 0,C 180,E1 -8736.497,E2 -8736.497} C_VEL
LIN {X 0,Y 445.885,Z 464.16,A -85,B 0,C 180,E1 -8738.155,E2 -8738.155} C_VEL
LIN {X 0,Y 446.24,Z 457.095,A -85,B 0,C 180,E1 -8739.519,E2 -8739.519} C_VEL
LIN {X 0,Y 446.685,Z 448.267,A -85,B 0,C 180,E1 -8740.883,E2 -8740.883} C_VEL
LIN {X 0,Y 447.253,Z 438.251,A -85,B 0,C 180,E1 -8742.132,E2 -8742.132} C_VEL
LIN {X 0,Y 447.845,Z 427.702,A -85,B 0,C 180,E1 -8743.195,E2 -8743.195} C_VEL
LIN {X 0,Y 448.344,Z 417.012,A -85,B 0,C 180,E1 -8744.062,E2 -8744.062} C_VEL
LIN {X 0,Y 448.976,Z 404.655,A -85,B 0,C 180,E1 -8744.852,E2 -8744.852} C_VEL
LIN {X 0,Y 449.381,Z 394.355,A -85,B 0,C 180,E1 -8745.361,E2 -8745.361} C_VEL
LIN {X 0,Y 447.36,Z 381.034,A -85,B 0,C 180,E1 -8745.925,E2 -8745.925} C_VEL
LIN {X 0,Y 446.143,Z 371.61,A -85,B 0,C 180,E1 -8746.218,E2 -8746.218} C_VEL
LIN {X 0,Y 446.456,Z 360.979,A -85,B 0,C 180,E1 -8749.304,E2 -8749.304} C_VEL
LIN {X 0,Y 446.846,Z 349.6,A -85,B 0,C 180,E1 -8752.665,E2 -8752.665} C_VEL
LIN {X 0,Y 447.194,Z 339.854,A -85,B 0,C 180,E1 -8755.606,E2 -8755.606} C_VEL
LIN {X 0,Y 447.579,Z 329.923,A -85,B 0,C 180,E1 -8758.727,E2 -8758.727} C_VEL
LIN {X 0,Y 448.078,Z 321.065,A -85,B 0,C 180,E1 -8761.651,E2 -8761.651} C_VEL
LIN {X 0,Y 448.737,Z 312.047,A -85,B 0,C 180,E1 -8764.866,E2 -8764.866} C_VEL
LIN {X 0,Y 448.924,Z 307.829,A -85,B 0,C 180,E1 -8766.506,E2 -8766.506} C_VEL
LIN {X 0,Y 448.122,Z 302.62,A -85,B 0,C 180,E1 -8768.854,E2 -8768.854} C_VEL
LIN {X 0,Y 447.239,Z 298.011,A -85,B 0,C 180,E1 -8771.3,E2 -8771.3} C_VEL
LIN {X 0,Y 446.439,Z 293.878,A -85,B 0,C 180,E1 -8774.155,E2 -8774.155} C_VEL
LIN {X 0,Y 446.423,Z 293.879,A -85,B 0,C 180,E1 -8777.725,E2 -8777.725} C_VEL
LIN {X 0,Y 446.439,Z 293.877,A -85,B 0,C 180,E1 -8780.972,E2 -8780.972} C_VEL
LIN {X 0,Y 446.422,Z 293.88,A -85,B 0,C 180,E1 -8784.374,E2 -8784.374} C_VEL
LIN {X 0,Y 446.425,Z 293.879,A -85,B 0,C 180,E1 -8787.639,E2 -8787.639} C_VEL
LIN {X 0,Y 446.451,Z 293.876,A -85,B 0,C 180,E1 -8790.791,E2 -8790.791} C_VEL
LIN {X 0,Y 446.465,Z 293.875,A -85,B 0,C 180,E1 -8792.838,E2 -8792.838} C_VEL
LIN {X 0,Y 446.585,Z 295.032,A -85,B 0,C 180,E1 -8794.855,E2 -8794.855} C_VEL
LIN {X 0,Y 446.586,Z 297.51,A -85,B 0,C 180,E1 -8798.202,E2 -8798.202} C_VEL
LIN {X 0,Y 446.542,Z 299.558,A -85,B 0,C 180,E1 -8800.792,E2 -8800.792} C_VEL
LIN {X 0,Y 446.412,Z 302.341,A -85,B 0,C 180,E1 -8804.139,E2 -8804.139} C_VEL
LIN {X 0,Y 449.843,Z 314.116,A -85,B 0,C 180,E1 -8804.714,E2 -8804.714} C_VEL
LIN {X 0,Y 449.481,Z 327.034,A -85,B 0,C 180,E1 -8805.339,E2 -8805.339} C_VEL
LIN {X 0,Y 449.1,Z 338.389,A -85,B 0,C 180,E1 -8806.069,E2 -8806.069} C_VEL
LIN {X 0,Y 448.617,Z 349.618,A -85,B 0,C 180,E1 -8806.985,E2 -8806.985} C_VEL
LIN {X 0,Y 448.121,Z 359.708,A -85,B 0,C 180,E1 -8808.006,E2 -8808.006} C_VEL
LIN {X 0,Y 447.595,Z 368.789,A -85,B 0,C 180,E1 -8809.139,E2 -8809.139} C_VEL
LIN {X 0,Y 447.135,Z 377.579,A -85,B 0,C 180,E1 -8810.501,E2 -8810.501} C_VEL
LIN {X 0,Y 446.726,Z 384.641,A -85,B 0,C 180,E1 -8811.86,E2 -8811.86} C_VEL
LIN {X 0,Y 446.449,Z 390.205,A -85,B 0,C 180,E1 -8813.22,E2 -8813.22} C_VEL
LIN {X 0,Y 446.13,Z 394.546,A -85,B 0,C 180,E1 -8814.576,E2 -8814.576} C_VEL
LIN {X 0,Y 446.124,Z 396.793,A -85,B 0,C 180,E1 -8815.482,E2 -8815.482} C_VEL
LIN {X 0,Y 445.924,Z 398.629,A -85,B 0,C 180,E1 -8816.386,E2 -8816.386} C_VEL
LIN {X 0,Y 445.727,Z 400.009,A -85,B 0,C 180,E1 -8817.289,E2 -8817.289} C_VEL
LIN {X 0,Y 445.582,Z 401.475,A -85,B 0,C 180,E1 -8819.096,E2 -8819.096} C_VEL
LIN {X 0,Y 445.563,Z 401.611,A -85,B 0,C 180,E1 -8820,E2 -8820} C_VEL
LIN {X 0,Y 445.561,Z 401.301,A -85,B 0,C 180,E1 -8820.904,E2 -8820.904} C_VEL
LIN {X 0,Y 445.711,Z 399.469,A -85,B 0,C 180,E1 -8822.711,E2 -8822.711} C_VEL
LIN {X 0,Y 445.958,Z 396.971,A -85,B 0,C 180,E1 -8824.067,E2 -8824.067} C_VEL
LIN {X 0,Y 446.036,Z 393.479,A -85,B 0,C 180,E1 -8825.425,E2 -8825.425} C_VEL
LIN {X 0,Y 446.177,Z 388.871,A -85,B 0,C 180,E1 -8826.786,E2 -8826.786} C_VEL
LIN {X 0,Y 446.506,Z 381.895,A -85,B 0,C 180,E1 -8828.372,E2 -8828.372} C_VEL
LIN {X 0,Y 446.889,Z 374.301,A -85,B 0,C 180,E1 -8829.733,E2 -8829.733} C_VEL
LIN {X 0,Y 447.249,Z 366.566,A -85,B 0,C 180,E1 -8830.869,E2 -8830.869} C_VEL
LIN {X 0,Y 447.759,Z 357.186,A -85,B 0,C 180,E1 -8832.004,E2 -8832.004} C_VEL
LIN {X 0,Y 448.297,Z 345.778,A -85,B 0,C 180,E1 -8833.112,E2 -8833.112} C_VEL
LIN {X 0,Y 448.652,Z 334.33,A -85,B 0,C 180,E1 -8834.006,E2 -8834.006} C_VEL
LIN {X 0,Y 449.107,Z 322.271,A -85,B 0,C 180,E1 -8834.732,E2 -8834.732} C_VEL
LIN {X 0,Y 449.218,Z 312.105,A -85,B 0,C 180,E1 -8835.213,E2 -8835.213} C_VEL
LIN {X 0,Y 446.051,Z 298.767,A -85,B 0,C 180,E1 -8835.777,E2 -8835.777} C_VEL
LIN {X 0,Y 445.807,Z 297.513,A -85,B 0,C 180,E1 -8835.825,E2 -8835.825} C_VEL
LIN {X 0,Y 445.784,Z 293.96,A -85,B 0,C 180,E1 -8838.927,E2 -8838.927} C_VEL
LIN {X 0,Y 446.134,Z 293.913,A -85,B 0,C 180,E1 -8842.215,E2 -8842.215} C_VEL
LIN {X 0,Y 446.395,Z 293.876,A -85,B 0,C 180,E1 -8845.156,E2 -8845.156} C_VEL
LIN {X 0,Y 446.488,Z 293.866,A -85,B 0,C 180,E1 -8848.179,E2 -8848.179} C_VEL
LIN {X 0,Y 446.421,Z 293.871,A -85,B 0,C 180,E1 -8851.775,E2 -8851.775} C_VEL
LIN {X 0,Y 446.432,Z 293.874,A -85,B 0,C 180,E1 -8854.523,E2 -8854.523} C_VEL
LIN {X 0,Y 446.419,Z 293.881,A -85,B 0,C 180,E1 -8858.079,E2 -8858.079} C_VEL
LIN {X 0,Y 446.43,Z 293.875,A -85,B 0,C 180,E1 -8860.918,E2 -8860.918} C_VEL
LIN {X 0,Y 446.42,Z 293.882,A -85,B 0,C 180,E1 -8863.844,E2 -8863.844} C_VEL
LIN {X 0,Y 446.402,Z 293.877,A -85,B 0,C 180,E1 -8866.403,E2 -8866.403} C_VEL
LIN {X 0,Y 446.429,Z 293.874,A -85,B 0,C 180,E1 -8869.082,E2 -8869.082} C_VEL
LIN {X 0,Y 446.412,Z 293.878,A -85,B 0,C 180,E1 -8872.121,E2 -8872.121} C_VEL
LIN {X 0,Y 446.347,Z 293.888,A -85,B 0,C 180,E1 -8874.962,E2 -8874.962} C_VEL
LIN {X 0,Y 446.182,Z 294.058,A -85,B 0,C 180,E1 -8876.767,E2 -8876.767} C_VEL
LIN {X 0,Y 445.972,Z 299.558,A -85,B 0,C 180,E1 -8880.082,E2 -8880.082} C_VEL
LIN {X 0,Y 445.913,Z 304.014,A -85,B 0,C 180,E1 -8882.802,E2 -8882.802} C_VEL
LIN {X 0,Y 445.856,Z 309.388,A -85,B 0,C 180,E1 -8886.1,E2 -8886.1} C_VEL
LIN {X 0,Y 445.842,Z 313.8,A -85,B 0,C 180,E1 -8888.742,E2 -8888.742} C_VEL
LIN {X 0,Y 445.777,Z 318.844,A -85,B 0,C 180,E1 -8891.62,E2 -8891.62} C_VEL
LIN {X 0,Y 445.813,Z 323.145,A -85,B 0,C 180,E1 -8893.936,E2 -8893.936} C_VEL
LIN {X 0,Y 448.979,Z 336.604,A -85,B 0,C 180,E1 -8894.443,E2 -8894.443} C_VEL
LIN {X 0,Y 449.778,Z 341.893,A -85,B 0,C 180,E1 -8894.682,E2 -8894.682} C_VEL
LIN {X 0,Y 449.413,Z 353.978,A -85,B 0,C 180,E1 -8895.278,E2 -8895.278} C_VEL
LIN {X 0,Y 448.872,Z 366.09,A -85,B 0,C 180,E1 -8896.078,E2 -8896.078} C_VEL
LIN {X 0,Y 448.395,Z 376.399,A -85,B 0,C 180,E1 -8896.944,E2 -8896.944} C_VEL
LIN {X 0,Y 447.501,Z 381.151,A -85,B 0,C 180,E1 -8897.38,E2 -8897.38} C_VEL
LIN {X 0,Y 444.294,Z 388.605,A -85,B 0,C 180,E1 -8898.114,E2 -8898.114} C_VEL
LIN {X 0,Y 441.033,Z 395.505,A -85,B 0,C 180,E1 -8898.935,E2 -8898.935} C_VEL
LIN {X 0,Y 440.066,Z 399.39,A -85,B 0,C 180,E1 -8899.501,E2 -8899.501} C_VEL
LIN {X 0,Y 439.579,Z 406.839,A -85,B 0,C 180,E1 -8900.8,E2 -8900.8} C_VEL
LIN {X 0,Y 439.182,Z 413.247,A -85,B 0,C 180,E1 -8902.182,E2 -8902.182} C_VEL
LIN {X 0,Y 438.945,Z 418.339,A -85,B 0,C 180,E1 -8903.565,E2 -8903.565} C_VEL
LIN {X 0,Y 438.647,Z 422.289,A -85,B 0,C 180,E1 -8904.944,E2 -8904.944} C_VEL
LIN {X 0,Y 438.612,Z 425.192,A -85,B 0,C 180,E1 -8906.325,E2 -8906.325} C_VEL
LIN {X 0,Y 438.519,Z 426.605,A -85,B 0,C 180,E1 -8907.244,E2 -8907.244} C_VEL
LIN {X 0,Y 438.373,Z 428.212,A -85,B 0,C 180,E1 -8909.081,E2 -8909.081} C_VEL
LIN {X 0,Y 438.349,Z 428.448,A -85,B 0,C 180,E1 -8910,E2 -8910} C_VEL
LIN {X 0,Y 438.451,Z 427.675,A -85,B 0,C 180,E1 -8911.837,E2 -8911.837} C_VEL
LIN {X 0,Y 438.608,Z 425.361,A -85,B 0,C 180,E1 -8913.675,E2 -8913.675} C_VEL
LIN {X 0,Y 438.606,Z 422.521,A -85,B 0,C 180,E1 -8915.056,E2 -8915.056} C_VEL
LIN {X 0,Y 438.946,Z 418.644,A -85,B 0,C 180,E1 -8916.435,E2 -8916.435} C_VEL
LIN {X 0,Y 439.142,Z 413.638,A -85,B 0,C 180,E1 -8917.818,E2 -8917.818} C_VEL
LIN {X 0,Y 439.562,Z 407.31,A -85,B 0,C 180,E1 -8919.2,E2 -8919.2} C_VEL
LIN {X 0,Y 440.071,Z 399.445,A -85,B 0,C 180,E1 -8920.583,E2 -8920.583} C_VEL
LIN {X 0,Y 440.644,Z 391.406,A -85,B 0,C 180,E1 -8921.733,E2 -8921.733} C_VEL
LIN {X 0,Y 441.233,Z 381.552,A -85,B 0,C 180,E1 -8922.885,E2 -8922.885} C_VEL
LIN {X 0,Y 441.787,Z 370.314,A -85,B 0,C 180,E1 -8923.934,E2 -8923.934} C_VEL
LIN {X 0,Y 442.366,Z 359.582,A -85,B 0,C 180,E1 -8924.726,E2 -8924.726} C_VEL
LIN {X 0,Y 442.852,Z 347.433,A -85,B 0,C 180,E1 -8925.416,E2 -8925.416} C_VEL
LIN {X 0,Y 442.711,Z 340.816,A -85,B 0,C 180,E1 -8925.723,E2 -8925.723} C_VEL
LIN {X 0,Y 439.994,Z 328.381,A -85,B 0,C 180,E1 -8926.257,E2 -8926.257} C_VEL
LIN {X 0,Y 438.745,Z 323.492,A -85,B 0,C 180,E1 -8926.432,E2 -8926.432} C_VEL
LIN {X 0,Y 438.73,Z 317.576,A -85,B 0,C 180,E1 -8929.658,E2 -8929.658} C_VEL
LIN {X 0,Y 438.785,Z 312.515,A -85,B 0,C 180,E1 -8932.607,E2 -8932.607} C_VEL
LIN {X 0,Y 438.825,Z 307.569,A -85,B 0,C 180,E1 -8935.621,E2 -8935.621} C_VEL
LIN {X 0,Y 438.862,Z 302.548,A -85,B 0,C 180,E1 -8938.713,E2 -8938.713} C_VEL
LIN {X 0,Y 439.018,Z 297.241,A -85,B 0,C 180,E1 -8941.956,E2 -8941.956} C_VEL
LIN {X 0,Y 439.164,Z 294.787,A -85,B 0,C 180,E1 -8943.501,E2 -8943.501} C_VEL
LIN {X 0,Y 439.362,Z 294.758,A -85,B 0,C 180,E1 -8946.289,E2 -8946.289} C_VEL
LIN {X 0,Y 439.404,Z 294.754,A -85,B 0,C 180,E1 -8949.849,E2 -8949.849} C_VEL
LIN {X 0,Y 439.384,Z 294.757,A -85,B 0,C 180,E1 -8952.627,E2 -8952.627} C_VEL
LIN {X 0,Y 439.402,Z 294.754,A -85,B 0,C 180,E1 -8955.271,E2 -8955.271} C_VEL
LIN {X 0,Y 439.391,Z 294.753,A -85,B 0,C 180,E1 -8958.743,E2 -8958.743} C_VEL
LIN {X 0,Y 439.379,Z 294.754,A -85,B 0,C 180,E1 -8961.607,E2 -8961.607} C_VEL
LIN {X 0,Y 439.314,Z 294.761,A -85,B 0,C 180,E1 -8964.836,E2 -8964.836} C_VEL
LIN {X 0,Y 439.067,Z 294.951,A -85,B 0,C 180,E1 -8967.028,E2 -8967.028} C_VEL
LIN {X 0,Y 438.918,Z 300.401,A -85,B 0,C 180,E1 -8970.239,E2 -8970.239} C_VEL
LIN {X 0,Y 438.836,Z 306.341,A -85,B 0,C 180,E1 -8973.747,E2 -8973.747} C_VEL
LIN {X 0,Y 438.778,Z 310.793,A -85,B 0,C 180,E1 -8976.395,E2 -8976.395} C_VEL
LIN {X 0,Y 438.738,Z 315.737,A -85,B 0,C 180,E1 -8979.365,E2 -8979.365} C_VEL
LIN {X 0,Y 438.696,Z 320.717,A -85,B 0,C 180,E1 -8982.279,E2 -8982.279} C_VEL
LIN {X 0,Y 438.707,Z 323.708,A -85,B 0,C 180,E1 -8984.033,E2 -8984.033} C_VEL
LIN {X 0,Y 441.863,Z 339.133,A -85,B 0,C 180,E1 -8984.667,E2 -8984.667} C_VEL
LIN {X 0,Y 442.199,Z 343.148,A -85,B 0,C 180,E1 -8984.856,E2 -8984.856} C_VEL
LIN {X 0,Y 441.733,Z 355.141,A -85,B 0,C 180,E1 -8985.488,E2 -8985.488} C_VEL
LIN {X 0,Y 441.203,Z 367.34,A -85,B 0,C 180,E1 -8986.333,E2 -8986.333} C_VEL
LIN {X 0,Y 440.795,Z 378.741,A -85,B 0,C 180,E1 -8987.336,E2 -8987.336} C_VEL
LIN {X 0,Y 440.214,Z 389.225,A -85,B 0,C 180,E1 -8988.489,E2 -8988.489} C_VEL
LIN {X 0,Y 439.783,Z 397.804,A -85,B 0,C 180,E1 -8989.643,E2 -8989.643} C_VEL
LIN {X 0,Y 439.412,Z 404.909,A -85,B 0,C 180,E1 -8990.796,E2 -8990.796} C_VEL
LIN {X 0,Y 439.057,Z 411.884,A -85,B 0,C 180,E1 -8992.18,E2 -8992.18} C_VEL
LIN {X 0,Y 438.87,Z 417.428,A -85,B 0,C 180,E1 -8993.564,E2 -8993.564} C_VEL
LIN {X 0,Y 438.579,Z 421.763,A -85,B 0,C 180,E1 -8994.944,E2 -8994.944} C_VEL
LIN {X 0,Y 438.609,Z 424.991,A -85,B 0,C 180,E1 -8996.325,E2 -8996.325} C_VEL
LIN {X 0,Y 438.519,Z 426.605,A -85,B 0,C 180,E1 -8997.244,E2 -8997.244} C_VEL
LIN {X 0,Y 438.452,Z 427.758,A -85,B 0,C 180,E1 -8998.163,E2 -8998.163} C_VEL
LIN {X 0,Y 438.352,Z 428.83,A -85,B 0,C 180,E1 -9000,E2 -9000} C_VEL
LIN {X 0,Y 438.376,Z 428.731,A -85,B 0,C 180,E1 -9000.919,E2 -9000.919} C_VEL
LIN {X 0,Y 438.472,Z 428.198,A -85,B 0,C 180,E1 -9001.837,E2 -9001.837} C_VEL
LIN {X 0,Y 438.603,Z 427.269,A -85,B 0,C 180,E1 -9002.755,E2 -9002.755} C_VEL
LIN {X 0,Y 438.626,Z 425.911,A -85,B 0,C 180,E1 -9003.675,E2 -9003.675} C_VEL
LIN {X 0,Y 438.705,Z 423.025,A -85,B 0,C 180,E1 -9005.055,E2 -9005.055} C_VEL
LIN {X 0,Y 438.944,Z 419.044,A -85,B 0,C 180,E1 -9006.435,E2 -9006.435} C_VEL
LIN {X 0,Y 439.252,Z 412.892,A -85,B 0,C 180,E1 -9008.048,E2 -9008.048} C_VEL
LIN {X 0,Y 439.685,Z 406.102,A -85,B 0,C 180,E1 -9009.43,E2 -9009.43} C_VEL
LIN {X 0,Y 440.152,Z 397.602,A -85,B 0,C 180,E1 -9010.814,E2 -9010.814} C_VEL
LIN {X 0,Y 440.671,Z 387.879,A -85,B 0,C 180,E1 -9012.083,E2 -9012.083} C_VEL
LIN {X 0,Y 441.297,Z 376.694,A -85,B 0,C 180,E1 -9013.25,E2 -9013.25} C_VEL
LIN {X 0,Y 441.751,Z 365.906,A -85,B 0,C 180,E1 -9014.147,E2 -9014.147} C_VEL
LIN {X 0,Y 442.306,Z 353.446,A -85,B 0,C 180,E1 -9014.963,E2 -9014.963} C_VEL
LIN {X 0,Y 442.751,Z 341.92,A -85,B 0,C 180,E1 -9015.537,E2 -9015.537} C_VEL
LIN {X 0,Y 440.369,Z 331.202,A -85,B 0,C 180,E1 -9016.055,E2 -9016.055} C_VEL
LIN {X 0,Y 439.008,Z 326.222,A -85,B 0,C 180,E1 -9016.285,E2 -9016.285} C_VEL
LIN {X 0,Y 439.041,Z 320.33,A -85,B 0,C 180,E1 -9019.643,E2 -9019.643} C_VEL
LIN {X 0,Y 439.069,Z 315.022,A -85,B 0,C 180,E1 -9022.592,E2 -9022.592} C_VEL
LIN {X 0,Y 439.064,Z 309.334,A -85,B 0,C 180,E1 -9025.606,E2 -9025.606} C_VEL
LIN {X 0,Y 439.183,Z 302.154,A -85,B 0,C 180,E1 -9029.214,E2 -9029.214} C_VEL
LIN {X 0,Y 439.202,Z 296.176,A -85,B 0,C 180,E1 -9031.995,E2 -9031.995} C_VEL
LIN {X 0,Y 439.158,Z 294.785,A -85,B 0,C 180,E1 -9032.696,E2 -9032.696} C_VEL
LIN {X 0,Y 439.36,Z 294.76,A -85,B 0,C 180,E1 -9035.334,E2 -9035.334} C_VEL
LIN {X 0,Y 439.379,Z 294.755,A -85,B 0,C 180,E1 -9038.596,E2 -9038.596} C_VEL
LIN {X 0,Y 439.383,Z 294.755,A -85,B 0,C 180,E1 -9041.256,E2 -9041.256} C_VEL
LIN {X 0,Y 439.402,Z 294.753,A -85,B 0,C 180,E1 -9044.729,E2 -9044.729} C_VEL
LIN {X 0,Y 439.403,Z 294.821,A -85,B 0,C 180,E1 -9046.997,E2 -9046.997} C_VEL
LIN {X 0,Y 441.069,Z 303.159,A -85,B 0,C 180,E1 -9050.405,E2 -9050.405} C_VEL
LIN {X 0,Y 442.177,Z 309.416,A -85,B 0,C 180,E1 -9052.845,E2 -9052.845} C_VEL
LIN {X 0,Y 442.351,Z 312.88,A -85,B 0,C 180,E1 -9054.123,E2 -9054.123} C_VEL
LIN {X 0,Y 441.694,Z 321.787,A -85,B 0,C 180,E1 -9057.249,E2 -9057.249} C_VEL
LIN {X 0,Y 441.097,Z 331.062,A -85,B 0,C 180,E1 -9060.401,E2 -9060.401} C_VEL
LIN {X 0,Y 440.431,Z 341.868,A -85,B 0,C 180,E1 -9063.971,E2 -9063.971} C_VEL
LIN {X 0,Y 440.065,Z 349.631,A -85,B 0,C 180,E1 -9066.468,E2 -9066.468} C_VEL
LIN {X 0,Y 439.645,Z 359.187,A -85,B 0,C 180,E1 -9069.41,E2 -9069.41} C_VEL
LIN {X 0,Y 439.222,Z 370.006,A -85,B 0,C 180,E1 -9072.781,E2 -9072.781} C_VEL
LIN {X 0,Y 439.154,Z 372.666,A -85,B 0,C 180,E1 -9073.541,E2 -9073.541} C_VEL
LIN {X 0,Y 441.153,Z 385.624,A -85,B 0,C 180,E1 -9073.979,E2 -9073.979} C_VEL
LIN {X 0,Y 442.537,Z 396.063,A -85,B 0,C 180,E1 -9074.455,E2 -9074.455} C_VEL
LIN {X 0,Y 441.965,Z 408.851,A -85,B 0,C 180,E1 -9075.142,E2 -9075.142} C_VEL
LIN {X 0,Y 441.313,Z 420.2,A -85,B 0,C 180,E1 -9075.945,E2 -9075.945} C_VEL
LIN {X 0,Y 440.699,Z 431.665,A -85,B 0,C 180,E1 -9076.971,E2 -9076.971} C_VEL
LIN {X 0,Y 440.158,Z 441.147,A -85,B 0,C 180,E1 -9078.02,E2 -9078.02} C_VEL
LIN {X 0,Y 439.567,Z 449.724,A -85,B 0,C 180,E1 -9079.172,E2 -9079.172} C_VEL
LIN {X 0,Y 439.141,Z 458.099,A -85,B 0,C 180,E1 -9080.558,E2 -9080.558} C_VEL
LIN {X 0,Y 438.752,Z 464.85,A -85,B 0,C 180,E1 -9081.943,E2 -9081.943} C_VEL
LIN {X 0,Y 438.545,Z 471.051,A -85,B 0,C 180,E1 -9083.559,E2 -9083.559} C_VEL
LIN {X 0,Y 438.44,Z 475.077,A -85,B 0,C 180,E1 -9084.942,E2 -9084.942} C_VEL
LIN {X 0,Y 438.333,Z 478.042,A -85,B 0,C 180,E1 -9086.323,E2 -9086.323} C_VEL
LIN {X 0,Y 438.353,Z 479.462,A -85,B 0,C 180,E1 -9087.243,E2 -9087.243} C_VEL
LIN {X 0,Y 438.342,Z 480.468,A -85,B 0,C 180,E1 -9088.162,E2 -9088.162} C_VEL
LIN {X 0,Y 438.315,Z 481.071,A -85,B 0,C 180,E1 -9089.081,E2 -9089.081} C_VEL
LIN {X 0,Y 438.29,Z 481.273,A -85,B 0,C 180,E1 -9090,E2 -9090} C_VEL
LIN {X 0,Y 438.315,Z 481.042,A -85,B 0,C 180,E1 -9090.919,E2 -9090.919} C_VEL
LIN {X 0,Y 438.359,Z 480.411,A -85,B 0,C 180,E1 -9091.838,E2 -9091.838} C_VEL
LIN {X 0,Y 438.354,Z 479.372,A -85,B 0,C 180,E1 -9092.757,E2 -9092.757} C_VEL
LIN {X 0,Y 438.349,Z 477.916,A -85,B 0,C 180,E1 -9093.677,E2 -9093.677} C_VEL
LIN {X 0,Y 438.443,Z 474.886,A -85,B 0,C 180,E1 -9095.058,E2 -9095.058} C_VEL
LIN {X 0,Y 438.546,Z 470.632,A -85,B 0,C 180,E1 -9096.488,E2 -9096.488} C_VEL
LIN {X 0,Y 438.754,Z 464.498,A -85,B 0,C 180,E1 -9098.057,E2 -9098.057} C_VEL
LIN {X 0,Y 439.141,Z 457.646,A -85,B 0,C 180,E1 -9099.442,E2 -9099.442} C_VEL
LIN {X 0,Y 439.564,Z 449.146,A -85,B 0,C 180,E1 -9100.828,E2 -9100.828} C_VEL
LIN {X 0,Y 440.118,Z 440.451,A -85,B 0,C 180,E1 -9101.981,E2 -9101.981} C_VEL
LIN {X 0,Y 440.743,Z 429.546,A -85,B 0,C 180,E1 -9103.155,E2 -9103.155} C_VEL
LIN {X 0,Y 441.245,Z 419.233,A -85,B 0,C 180,E1 -9104.058,E2 -9104.058} C_VEL
LIN {X 0,Y 441.851,Z 407.782,A -85,B 0,C 180,E1 -9104.861,E2 -9104.861} C_VEL
LIN {X 0,Y 442.422,Z 394.858,A -85,B 0,C 180,E1 -9105.549,E2 -9105.549} C_VEL
LIN {X 0,Y 440.318,Z 380.784,A -85,B 0,C 180,E1 -9106.174,E2 -9106.174} C_VEL
LIN {X 0,Y 439.09,Z 370.839,A -85,B 0,C 180,E1 -9106.497,E2 -9106.497} C_VEL
LIN {X 0,Y 439.401,Z 360.292,A -85,B 0,C 180,E1 -9109.626,E2 -9109.626} C_VEL
LIN {X 0,Y 439.81,Z 348.943,A -85,B 0,C 180,E1 -9113.048,E2 -9113.048} C_VEL
LIN {X 0,Y 440.194,Z 339.298,A -85,B 0,C 180,E1 -9116.044,E2 -9116.044} C_VEL
LIN {X 0,Y 440.76,Z 328.259,A -85,B 0,C 180,E1 -9119.624,E2 -9119.624} C_VEL
LIN {X 0,Y 441.28,Z 319.13,A -85,B 0,C 180,E1 -9122.786,E2 -9122.786} C_VEL
LIN {X 0,Y 441.897,Z 312.227,A -85,B 0,C 180,E1 -9125.368,E2 -9125.368} C_VEL
LIN {X 0,Y 441.832,Z 307.837,A -85,B 0,C 180,E1 -9127.189,E2 -9127.189} C_VEL
LIN {X 0,Y 440.821,Z 301.988,A -85,B 0,C 180,E1 -9130.069,E2 -9130.069} C_VEL
LIN {X 0,Y 439.922,Z 297.677,A -85,B 0,C 180,E1 -9132.703,E2 -9132.703} C_VEL
LIN {X 0,Y 439.41,Z 294.753,A -85,B 0,C 180,E1 -9135.133,E2 -9135.133} C_VEL
LIN {X 0,Y 439.383,Z 294.756,A -85,B 0,C 180,E1 -9138.744,E2 -9138.744} C_VEL
LIN {X 0,Y 439.374,Z 294.756,A -85,B 0,C 180,E1 -9141.608,E2 -9141.608} C_VEL
LIN {X 0,Y 439.402,Z 294.752,A -85,B 0,C 180,E1 -9144.844,E2 -9144.844} C_VEL
LIN {X 0,Y 439.376,Z 294.757,A -85,B 0,C 180,E1 -9148.14,E2 -9148.14} C_VEL
LIN {X 0,Y 439.435,Z 294.751,A -85,B 0,C 180,E1 -9151.598,E2 -9151.598} C_VEL
LIN {X 0,Y 439.438,Z 294.75,A -85,B 0,C 180,E1 -9152.367,E2 -9152.367} C_VEL
LIN {X 0,Y 439.628,Z 296.92,A -85,B 0,C 180,E1 -9155.674,E2 -9155.674} C_VEL
LIN {X 0,Y 439.582,Z 298.942,A -85,B 0,C 180,E1 -9158.425,E2 -9158.425} C_VEL
LIN {X 0,Y 439.481,Z 301.212,A -85,B 0,C 180,E1 -9161.347,E2 -9161.347} C_VEL
LIN {X 0,Y 439.418,Z 303.259,A -85,B 0,C 180,E1 -9163.845,E2 -9163.845} C_VEL
LIN {X 0,Y 442.731,Z 314.004,A -85,B 0,C 180,E1 -9164.388,E2 -9164.388} C_VEL
LIN {X 0,Y 443.048,Z 316.939,A -85,B 0,C 180,E1 -9164.532,E2 -9164.532} C_VEL
LIN {X 0,Y 442.671,Z 329.202,A -85,B 0,C 180,E1 -9165.167,E2 -9165.167} C_VEL
LIN {X 0,Y 442.156,Z 341.902,A -85,B 0,C 180,E1 -9166.039,E2 -9166.039} C_VEL
LIN {X 0,Y 441.663,Z 353.011,A -85,B 0,C 180,E1 -9167.011,E2 -9167.011} C_VEL
LIN {X 0,Y 441.126,Z 362.575,A -85,B 0,C 180,E1 -9168.047,E2 -9168.047} C_VEL
LIN {X 0,Y 440.609,Z 371.286,A -85,B 0,C 180,E1 -9169.198,E2 -9169.198} C_VEL
LIN {X 0,Y 440.137,Z 379.748,A -85,B 0,C 180,E1 -9170.58,E2 -9170.58} C_VEL
LIN {X 0,Y 439.701,Z 386.56,A -85,B 0,C 180,E1 -9171.984,E2 -9171.984} C_VEL
LIN {X 0,Y 439.24,Z 392.584,A -85,B 0,C 180,E1 -9173.569,E2 -9173.569} C_VEL
LIN {X 0,Y 439.117,Z 396.52,A -85,B 0,C 180,E1 -9174.95,E2 -9174.95} C_VEL
LIN {X 0,Y 438.89,Z 399.392,A -85,B 0,C 180,E1 -9176.328,E2 -9176.328} C_VEL
LIN {X 0,Y 438.68,Z 400.756,A -85,B 0,C 180,E1 -9177.245,E2 -9177.245} C_VEL
LIN {X 0,Y 438.567,Z 401.677,A -85,B 0,C 180,E1 -9178.163,E2 -9178.163} C_VEL
LIN {X 0,Y 438.52,Z 402.195,A -85,B 0,C 180,E1 -9179.082,E2 -9179.082} C_VEL
LIN {X 0,Y 438.498,Z 402.31,A -85,B 0,C 180,E1 -9180,E2 -9180} C_VEL
LIN {X 0,Y 438.494,Z 401.978,A -85,B 0,C 180,E1 -9180.918,E2 -9180.918} C_VEL
LIN {X 0,Y 438.53,Z 401.244,A -85,B 0,C 180,E1 -9181.837,E2 -9181.837} C_VEL
LIN {X 0,Y 438.665,Z 400.101,A -85,B 0,C 180,E1 -9182.755,E2 -9182.755} C_VEL
LIN {X 0,Y 438.924,Z 397.564,A -85,B 0,C 180,E1 -9184.132,E2 -9184.132} C_VEL
LIN {X 0,Y 438.991,Z 394.029,A -85,B 0,C 180,E1 -9185.512,E2 -9185.512} C_VEL
LIN {X 0,Y 439.189,Z 388.771,A -85,B 0,C 180,E1 -9187.044,E2 -9187.044} C_VEL
LIN {X 0,Y 439.5,Z 382.319,A -85,B 0,C 180,E1 -9188.506,E2 -9188.506} C_VEL
LIN {X 0,Y 439.902,Z 374.665,A -85,B 0,C 180,E1 -9189.889,E2 -9189.889} C_VEL
LIN {X 0,Y 440.289,Z 366.861,A -85,B 0,C 180,E1 -9191.043,E2 -9191.043} C_VEL
LIN {X 0,Y 440.823,Z 357.371,A -85,B 0,C 180,E1 -9192.195,E2 -9192.195} C_VEL
LIN {X 0,Y 441.369,Z 346.177,A -85,B 0,C 180,E1 -9193.294,E2 -9193.294} C_VEL
LIN {X 0,Y 441.718,Z 335.271,A -85,B 0,C 180,E1 -9194.159,E2 -9194.159} C_VEL
LIN {X 0,Y 442.211,Z 323.132,A -85,B 0,C 180,E1 -9194.908,E2 -9194.908} C_VEL
LIN {X 0,Y 442.27,Z 313.146,A -85,B 0,C 180,E1 -9195.396,E2 -9195.396} C_VEL
LIN {X 0,Y 439.054,Z 299.613,A -85,B 0,C 180,E1 -9195.979,E2 -9195.979} C_VEL
LIN {X 0,Y 438.72,Z 298.025,A -85,B 0,C 180,E1 -9196.065,E2 -9196.065} C_VEL
LIN {X 0,Y 438.706,Z 294.88,A -85,B 0,C 180,E1 -9198.687,E2 -9198.687} C_VEL
LIN {X 0,Y 439.046,Z 294.795,A -85,B 0,C 180,E1 -9201.808,E2 -9201.808} C_VEL
LIN {X 0,Y 439.309,Z 294.766,A -85,B 0,C 180,E1 -9204.579,E2 -9204.579} C_VEL
LIN {X 0,Y 439.413,Z 294.745,A -85,B 0,C 180,E1 -9207.635,E2 -9207.635} C_VEL
LIN {X 0,Y 439.364,Z 294.752,A -85,B 0,C 180,E1 -9210.788,E2 -9210.788} C_VEL
LIN {X 0,Y 439.39,Z 294.754,A -85,B 0,C 180,E1 -9214.044,E2 -9214.044} C_VEL
LIN {X 0,Y 439.351,Z 294.758,A -85,B 0,C 180,E1 -9216.887,E2 -9216.887} C_VEL
LIN {X 0,Y 439.404,Z 294.752,A -85,B 0,C 180,E1 -9219.849,E2 -9219.849} C_VEL
LIN {X 0,Y 439.385,Z 294.753,A -85,B 0,C 180,E1 -9222.627,E2 -9222.627} C_VEL
LIN {X 0,Y 439.404,Z 294.749,A -85,B 0,C 180,E1 -9225.271,E2 -9225.271} C_VEL
LIN {X 0,Y 439.391,Z 294.75,A -85,B 0,C 180,E1 -9228.743,E2 -9228.743} C_VEL
LIN {X 0,Y 439.377,Z 294.757,A -85,B 0,C 180,E1 -9231.608,E2 -9231.608} C_VEL
LIN {X 0,Y 439.332,Z 294.762,A -85,B 0,C 180,E1 -9234.838,E2 -9234.838} C_VEL
LIN {X 0,Y 439.136,Z 294.983,A -85,B 0,C 180,E1 -9236.795,E2 -9236.795} C_VEL
LIN {X 0,Y 438.916,Z 300.679,A -85,B 0,C 180,E1 -9240.239,E2 -9240.239} C_VEL
LIN {X 0,Y 438.864,Z 306.359,A -85,B 0,C 180,E1 -9243.74,E2 -9243.74} C_VEL
LIN {X 0,Y 438.795,Z 310.695,A -85,B 0,C 180,E1 -9246.396,E2 -9246.396} C_VEL
LIN {X 0,Y 438.758,Z 315.699,A -85,B 0,C 180,E1 -9249.366,E2 -9249.366} C_VEL
LIN {X 0,Y 438.712,Z 320.882,A -85,B 0,C 180,E1 -9252.279,E2 -9252.279} C_VEL
LIN {X 0,Y 438.744,Z 323.485,A -85,B 0,C 180,E1 -9253.663,E2 -9253.663} C_VEL
LIN {X 0,Y 441.968,Z 337.21,A -85,B 0,C 180,E1 -9254.197,E2 -9254.197} C_VEL
LIN {X 0,Y 442.966,Z 342.986,A -85,B 0,C 180,E1 -9254.47,E2 -9254.47} C_VEL
LIN {X 0,Y 442.559,Z 354.377,A -85,B 0,C 180,E1 -9255.045,E2 -9255.045} C_VEL
LIN {X 0,Y 442,Z 366.416,A -85,B 0,C 180,E1 -9255.851,E2 -9255.851} C_VEL
LIN {X 0,Y 441.489,Z 377.184,A -85,B 0,C 180,E1 -9256.772,E2 -9256.772} C_VEL
LIN {X 0,Y 440.929,Z 386.941,A -85,B 0,C 180,E1 -9257.808,E2 -9257.808} C_VEL
LIN {X 0,Y 440.333,Z 395.772,A -85,B 0,C 180,E1 -9258.958,E2 -9258.958} C_VEL
LIN {X 0,Y 440.066,Z 399.39,A -85,B 0,C 180,E1 -9259.501,E2 -9259.501} C_VEL
LIN {X 0,Y 439.108,Z 403.128,A -85,B 0,C 180,E1 -9260.092,E2 -9260.092} C_VEL
LIN {X 0,Y 435.884,Z 408.811,A -85,B 0,C 180,E1 -9261.073,E2 -9261.073} C_VEL
LIN {X 0,Y 432.768,Z 413.854,A -85,B 0,C 180,E1 -9262.121,E2 -9262.121} C_VEL
LIN {X 0,Y 431.984,Z 416.521,A -85,B 0,C 180,E1 -9262.806,E2 -9262.806} C_VEL
LIN {X 0,Y 431.757,Z 420.173,A -85,B 0,C 180,E1 -9263.926,E2 -9263.926} C_VEL
LIN {X 0,Y 431.605,Z 423.76,A -85,B 0,C 180,E1 -9265.33,E2 -9265.33} C_VEL
LIN {X 0,Y 431.555,Z 425.607,A -85,B 0,C 180,E1 -9266.265,E2 -9266.265} C_VEL
LIN {X 0,Y 431.447,Z 427.02,A -85,B 0,C 180,E1 -9267.199,E2 -9267.199} C_VEL
LIN {X 0,Y 431.314,Z 428.626,A -85,B 0,C 180,E1 -9269.066,E2 -9269.066} C_VEL
LIN {X 0,Y 431.288,Z 428.861,A -85,B 0,C 180,E1 -9270,E2 -9270} C_VEL
LIN {X 0,Y 431.314,Z 428.672,A -85,B 0,C 180,E1 -9270.934,E2 -9270.934} C_VEL
LIN {X 0,Y 431.447,Z 427.128,A -85,B 0,C 180,E1 -9272.801,E2 -9272.801} C_VEL
LIN {X 0,Y 431.55,Z 425.774,A -85,B 0,C 180,E1 -9273.735,E2 -9273.735} C_VEL
LIN {X 0,Y 431.534,Z 422.935,A -85,B 0,C 180,E1 -9275.139,E2 -9275.139} C_VEL
LIN {X 0,Y 431.906,Z 419.056,A -85,B 0,C 180,E1 -9276.54,E2 -9276.54} C_VEL
LIN {X 0,Y 432.128,Z 414.048,A -85,B 0,C 180,E1 -9277.946,E2 -9277.946} C_VEL
LIN {X 0,Y 432.557,Z 407.72,A -85,B 0,C 180,E1 -9279.351,E2 -9279.351} C_VEL
LIN {X 0,Y 433.111,Z 399.851,A -85,B 0,C 180,E1 -9280.755,E2 -9280.755} C_VEL
LIN {X 0,Y 433.707,Z 391.81,A -85,B 0,C 180,E1 -9281.924,E2 -9281.924} C_VEL
LIN {X 0,Y 434.344,Z 381.95,A -85,B 0,C 180,E1 -9283.093,E2 -9283.093} C_VEL
LIN {X 0,Y 434.911,Z 370.603,A -85,B 0,C 180,E1 -9284.168,E2 -9284.168} C_VEL
LIN {X 0,Y 435.539,Z 359.968,A -85,B 0,C 180,E1 -9284.962,E2 -9284.962} C_VEL
LIN {X 0,Y 436.02,Z 347.805,A -85,B 0,C 180,E1 -9285.663,E2 -9285.663} C_VEL
LIN {X 0,Y 435.899,Z 341.996,A -85,B 0,C 180,E1 -9285.941,E2 -9285.941} C_VEL
LIN {X 0,Y 433.275,Z 329.995,A -85,B 0,C 180,E1 -9286.478,E2 -9286.478} C_VEL
LIN {X 0,Y 431.697,Z 323.855,A -85,B 0,C 180,E1 -9286.704,E2 -9286.704} C_VEL
LIN {X 0,Y 431.691,Z 317.843,A -85,B 0,C 180,E1 -9289.992,E2 -9289.992} C_VEL
LIN {X 0,Y 431.738,Z 312.712,A -85,B 0,C 180,E1 -9292.997,E2 -9292.997} C_VEL
LIN {X 0,Y 431.802,Z 307.057,A -85,B 0,C 180,E1 -9296.468,E2 -9296.468} C_VEL
LIN {X 0,Y 431.83,Z 302.577,A -85,B 0,C 180,E1 -9299.226,E2 -9299.226} C_VEL
LIN {X 0,Y 432.046,Z 296.361,A -85,B 0,C 180,E1 -9303.021,E2 -9303.021} C_VEL
LIN {X 0,Y 432.14,Z 295.662,A -85,B 0,C 180,E1 -9303.57,E2 -9303.57} C_VEL
LIN {X 0,Y 432.315,Z 295.638,A -85,B 0,C 180,E1 -9305.82,E2 -9305.82} C_VEL
LIN {X 0,Y 432.349,Z 295.631,A -85,B 0,C 180,E1 -9309.343,E2 -9309.343} C_VEL
LIN {X 0,Y 432.336,Z 295.632,A -85,B 0,C 180,E1 -9311.797,E2 -9311.797} C_VEL
LIN {X 0,Y 432.336,Z 295.633,A -85,B 0,C 180,E1 -9314.347,E2 -9314.347} C_VEL
LIN {X 0,Y 432.322,Z 295.634,A -85,B 0,C 180,E1 -9317.016,E2 -9317.016} C_VEL
LIN {X 0,Y 432.344,Z 295.631,A -85,B 0,C 180,E1 -9319.82,E2 -9319.82} C_VEL
LIN {X 0,Y 432.3,Z 295.638,A -85,B 0,C 180,E1 -9323.021,E2 -9323.021} C_VEL
LIN {X 0,Y 432.154,Z 295.655,A -85,B 0,C 180,E1 -9326.037,E2 -9326.037} C_VEL
LIN {X 0,Y 432.013,Z 295.702,A -85,B 0,C 180,E1 -9326.977,E2 -9326.977} C_VEL
LIN {X 0,Y 431.832,Z 302.111,A -85,B 0,C 180,E1 -9330.774,E2 -9330.774} C_VEL
LIN {X 0,Y 431.768,Z 307.406,A -85,B 0,C 180,E1 -9333.929,E2 -9333.929} C_VEL
LIN {X 0,Y 431.712,Z 312.577,A -85,B 0,C 180,E1 -9337.001,E2 -9337.001} C_VEL
LIN {X 0,Y 431.651,Z 317.582,A -85,B 0,C 180,E1 -9340.006,E2 -9340.006} C_VEL
LIN {X 0,Y 431.628,Z 322.57,A -85,B 0,C 180,E1 -9342.957,E2 -9342.957} C_VEL
LIN {X 0,Y 431.638,Z 324.047,A -85,B 0,C 180,E1 -9343.831,E2 -9343.831} C_VEL
LIN {X 0,Y 434.516,Z 337.806,A -85,B 0,C 180,E1 -9344.385,E2 -9344.385} C_VEL
LIN {X 0,Y 435.285,Z 343.669,A -85,B 0,C 180,E1 -9344.669,E2 -9344.669} C_VEL
LIN {X 0,Y 434.746,Z 356.554,A -85,B 0,C 180,E1 -9345.369,E2 -9345.369} C_VEL
LIN {X 0,Y 434.182,Z 369.075,A -85,B 0,C 180,E1 -9346.273,E2 -9346.273} C_VEL
LIN {X 0,Y 433.78,Z 379.761,A -85,B 0,C 180,E1 -9347.247,E2 -9347.247} C_VEL
LIN {X 0,Y 433.224,Z 389.192,A -85,B 0,C 180,E1 -9348.3,E2 -9348.3} C_VEL
LIN {X 0,Y 432.769,Z 397.852,A -85,B 0,C 180,E1 -9349.473,E2 -9349.473} C_VEL
LIN {X 0,Y 432.304,Z 406.328,A -85,B 0,C 180,E1 -9350.88,E2 -9350.88} C_VEL
LIN {X 0,Y 431.96,Z 413.095,A -85,B 0,C 180,E1 -9352.286,E2 -9352.286} C_VEL
LIN {X 0,Y 431.787,Z 417.692,A -85,B 0,C 180,E1 -9353.458,E2 -9353.458} C_VEL
LIN {X 0,Y 431.512,Z 422.075,A -85,B 0,C 180,E1 -9354.861,E2 -9354.861} C_VEL
LIN {X 0,Y 431.553,Z 425.347,A -85,B 0,C 180,E1 -9356.265,E2 -9356.265} C_VEL
LIN {X 0,Y 431.447,Z 426.985,A -85,B 0,C 180,E1 -9357.199,E2 -9357.199} C_VEL
LIN {X 0,Y 431.368,Z 428.171,A -85,B 0,C 180,E1 -9358.133,E2 -9358.133} C_VEL
LIN {X 0,Y 431.316,Z 428.919,A -85,B 0,C 180,E1 -9359.066,E2 -9359.066} C_VEL
LIN {X 0,Y 431.291,Z 429.275,A -85,B 0,C 180,E1 -9360,E2 -9360} C_VEL
LIN {X 0,Y 431.318,Z 429.2,A -85,B 0,C 180,E1 -9360.934,E2 -9360.934} C_VEL
LIN {X 0,Y 431.419,Z 428.678,A -85,B 0,C 180,E1 -9361.867,E2 -9361.867} C_VEL
LIN {X 0,Y 431.524,Z 427.76,A -85,B 0,C 180,E1 -9362.801,E2 -9362.801} C_VEL
LIN {X 0,Y 431.571,Z 426.416,A -85,B 0,C 180,E1 -9363.735,E2 -9363.735} C_VEL
LIN {X 0,Y 431.658,Z 423.551,A -85,B 0,C 180,E1 -9365.138,E2 -9365.138} C_VEL
LIN {X 0,Y 431.92,Z 419.594,A -85,B 0,C 180,E1 -9366.54,E2 -9366.54} C_VEL
LIN {X 0,Y 432.241,Z 413.476,A -85,B 0,C 180,E1 -9368.179,E2 -9368.179} C_VEL
LIN {X 0,Y 432.72,Z 406.703,A -85,B 0,C 180,E1 -9369.583,E2 -9369.583} C_VEL
LIN {X 0,Y 433.215,Z 398.207,A -85,B 0,C 180,E1 -9370.989,E2 -9370.989} C_VEL
LIN {X 0,Y 433.657,Z 389.502,A -85,B 0,C 180,E1 -9372.162,E2 -9372.162} C_VEL
LIN {X 0,Y 434.313,Z 379.305,A -85,B 0,C 180,E1 -9373.276,E2 -9373.276} C_VEL
LIN {X 0,Y 434.847,Z 368.412,A -85,B 0,C 180,E1 -9374.245,E2 -9374.245} C_VEL
LIN {X 0,Y 435.395,Z 356.313,A -85,B 0,C 180,E1 -9375.087,E2 -9375.087} C_VEL
LIN {X 0,Y 435.984,Z 343.086,A -85,B 0,C 180,E1 -9375.785,E2 -9375.785} C_VEL
LIN {X 0,Y 433.36,Z 331.622,A -85,B 0,C 180,E1 -9376.359,E2 -9376.359} C_VEL
LIN {X 0,Y 431.995,Z 326.774,A -85,B 0,C 180,E1 -9376.602,E2 -9376.602} C_VEL
LIN {X 0,Y 432.032,Z 320.882,A -85,B 0,C 180,E1 -9379.975,E2 -9379.975} C_VEL
LIN {X 0,Y 432.044,Z 315.47,A -85,B 0,C 180,E1 -9382.98,E2 -9382.98} C_VEL
LIN {X 0,Y 432.056,Z 309.712,A -85,B 0,C 180,E1 -9386.052,E2 -9386.052} C_VEL
LIN {X 0,Y 432.195,Z 302.389,A -85,B 0,C 180,E1 -9389.734,E2 -9389.734} C_VEL
LIN {X 0,Y 432.177,Z 296.004,A -85,B 0,C 180,E1 -9392.732,E2 -9392.732} C_VEL
LIN {X 0,Y 432.173,Z 295.655,A -85,B 0,C 180,E1 -9393.009,E2 -9393.009} C_VEL
LIN {X 0,Y 432.326,Z 295.635,A -85,B 0,C 180,E1 -9395.819,E2 -9395.819} C_VEL
LIN {X 0,Y 432.33,Z 295.634,A -85,B 0,C 180,E1 -9399.345,E2 -9399.345} C_VEL
LIN {X 0,Y 432.326,Z 295.634,A -85,B 0,C 180,E1 -9401.798,E2 -9401.798} C_VEL
LIN {X 0,Y 432.336,Z 295.633,A -85,B 0,C 180,E1 -9404.347,E2 -9404.347} C_VEL
LIN {X 0,Y 432.346,Z 295.632,A -85,B 0,C 180,E1 -9406.614,E2 -9406.614} C_VEL
LIN {X 0,Y 433.749,Z 302.79,A -85,B 0,C 180,E1 -9409.6,E2 -9409.6} C_VEL
LIN {X 0,Y 435.026,Z 309.624,A -85,B 0,C 180,E1 -9412.337,E2 -9412.337} C_VEL
LIN {X 0,Y 435.435,Z 313.478,A -85,B 0,C 180,E1 -9413.805,E2 -9413.805} C_VEL
LIN {X 0,Y 434.804,Z 321.478,A -85,B 0,C 180,E1 -9416.663,E2 -9416.663} C_VEL
LIN {X 0,Y 434.185,Z 330.739,A -85,B 0,C 180,E1 -9419.882,E2 -9419.882} C_VEL
LIN {X 0,Y 433.56,Z 340.189,A -85,B 0,C 180,E1 -9423.069,E2 -9423.069} C_VEL
LIN {X 0,Y 433.107,Z 349.275,A -85,B 0,C 180,E1 -9426.067,E2 -9426.067} C_VEL
LIN {X 0,Y 432.568,Z 360.259,A -85,B 0,C 180,E1 -9429.555,E2 -9429.555} C_VEL
LIN {X 0,Y 432.121,Z 371.075,A -85,B 0,C 180,E1 -9432.977,E2 -9432.977} C_VEL
LIN {X 0,Y 432.094,Z 372.119,A -85,B 0,C 180,E1 -9433.259,E2 -9433.259} C_VEL
LIN {X 0,Y 434.263,Z 386.487,A -85,B 0,C 180,E1 -9433.766,E2 -9433.766} C_VEL
LIN {X 0,Y 435.635,Z 396.767,A -85,B 0,C 180,E1 -9434.262,E2 -9434.262} C_VEL
LIN {X 0,Y 435.079,Z 408.288,A -85,B 0,C 180,E1 -9434.902,E2 -9434.902} C_VEL
LIN {X 0,Y 434.393,Z 419.621,A -85,B 0,C 180,E1 -9435.716,E2 -9435.716} C_VEL
LIN {X 0,Y 433.731,Z 430.832,A -85,B 0,C 180,E1 -9436.734,E2 -9436.734} C_VEL
LIN {X 0,Y 433.162,Z 440.55,A -85,B 0,C 180,E1 -9437.823,E2 -9437.823} C_VEL
LIN {X 0,Y 432.547,Z 449.133,A -85,B 0,C 180,E1 -9438.994,E2 -9438.994} C_VEL
LIN {X 0,Y 432.082,Z 457.51,A -85,B 0,C 180,E1 -9440.403,E2 -9440.403} C_VEL
LIN {X 0,Y 431.711,Z 464.265,A -85,B 0,C 180,E1 -9441.811,E2 -9441.811} C_VEL
LIN {X 0,Y 431.479,Z 470.633,A -85,B 0,C 180,E1 -9443.505,E2 -9443.505} C_VEL
LIN {X 0,Y 431.377,Z 474.499,A -85,B 0,C 180,E1 -9444.859,E2 -9444.859} C_VEL
LIN {X 0,Y 431.245,Z 477.462,A -85,B 0,C 180,E1 -9446.262,E2 -9446.262} C_VEL
LIN {X 0,Y 431.284,Z 478.883,A -85,B 0,C 180,E1 -9447.198,E2 -9447.198} C_VEL
LIN {X 0,Y 431.262,Z 479.886,A -85,B 0,C 180,E1 -9448.132,E2 -9448.132} C_VEL
LIN {X 0,Y 431.259,Z 480.486,A -85,B 0,C 180,E1 -9449.066,E2 -9449.066} C_VEL
LIN {X 0,Y 431.233,Z 480.684,A -85,B 0,C 180,E1 -9450,E2 -9450} C_VEL
LIN {X 0,Y 431.259,Z 480.447,A -85,B 0,C 180,E1 -9450.934,E2 -9450.934} C_VEL
LIN {X 0,Y 431.291,Z 479.809,A -85,B 0,C 180,E1 -9451.868,E2 -9451.868} C_VEL
LIN {X 0,Y 431.285,Z 478.756,A -85,B 0,C 180,E1 -9452.802,E2 -9452.802} C_VEL
LIN {X 0,Y 431.263,Z 477.29,A -85,B 0,C 180,E1 -9453.738,E2 -9453.738} C_VEL
LIN {X 0,Y 431.383,Z 474.243,A -85,B 0,C 180,E1 -9455.141,E2 -9455.141} C_VEL
LIN {X 0,Y 431.482,Z 470.123,A -85,B 0,C 180,E1 -9456.547,E2 -9456.547} C_VEL
LIN {X 0,Y 431.716,Z 463.809,A -85,B 0,C 180,E1 -9458.189,E2 -9458.189} C_VEL
LIN {X 0,Y 432.082,Z 456.921,A -85,B 0,C 180,E1 -9459.597,E2 -9459.597} C_VEL
LIN {X 0,Y 432.546,Z 448.399,A -85,B 0,C 180,E1 -9461.006,E2 -9461.006} C_VEL
LIN {X 0,Y 433.082,Z 439.672,A -85,B 0,C 180,E1 -9462.179,E2 -9462.179} C_VEL
LIN {X 0,Y 433.711,Z 429.844,A -85,B 0,C 180,E1 -9463.263,E2 -9463.263} C_VEL
LIN {X 0,Y 434.308,Z 418.431,A -85,B 0,C 180,E1 -9464.287,E2 -9464.287} C_VEL
LIN {X 0,Y 434.954,Z 406.98,A -85,B 0,C 180,E1 -9465.103,E2 -9465.103} C_VEL
LIN {X 0,Y 435.441,Z 395.358,A -85,B 0,C 180,E1 -9465.745,E2 -9465.745} C_VEL
LIN {X 0,Y 433.39,Z 380.872,A -85,B 0,C 180,E1 -9466.417,E2 -9466.417} C_VEL
LIN {X 0,Y 432.052,Z 370.09,A -85,B 0,C 180,E1 -9466.786,E2 -9466.786} C_VEL
LIN {X 0,Y 432.347,Z 359.602,A -85,B 0,C 180,E1 -9469.96,E2 -9469.96} C_VEL
LIN {X 0,Y 432.787,Z 348.338,A -85,B 0,C 180,E1 -9473.444,E2 -9473.444} C_VEL
LIN {X 0,Y 433.265,Z 337.677,A -85,B 0,C 180,E1 -9476.854,E2 -9476.854} C_VEL
LIN {X 0,Y 433.888,Z 326.83,A -85,B 0,C 180,E1 -9480.507,E2 -9480.507} C_VEL
LIN {X 0,Y 434.508,Z 317.463,A -85,B 0,C 180,E1 -9483.919,E2 -9483.919} C_VEL
LIN {X 0,Y 435.075,Z 311.879,A -85,B 0,C 180,E1 -9486.13,E2 -9486.13} C_VEL
LIN {X 0,Y 434.675,Z 307.93,A -85,B 0,C 180,E1 -9487.909,E2 -9487.909} C_VEL
LIN {X 0,Y 433.833,Z 303.147,A -85,B 0,C 180,E1 -9490.413,E2 -9490.413} C_VEL
LIN {X 0,Y 433,Z 299.024,A -85,B 0,C 180,E1 -9493.08,E2 -9493.08} C_VEL
LIN {X 0,Y 432.409,Z 296.034,A -85,B 0,C 180,E1 -9495.662,E2 -9495.662} C_VEL
LIN {X 0,Y 432.309,Z 295.638,A -85,B 0,C 180,E1 -9496.297,E2 -9496.297} C_VEL
LIN {X 0,Y 432.323,Z 295.636,A -85,B 0,C 180,E1 -9499.439,E2 -9499.439} C_VEL
LIN {X 0,Y 432.337,Z 295.634,A -85,B 0,C 180,E1 -9501.85,E2 -9501.85} C_VEL
LIN {X 0,Y 432.342,Z 295.633,A -85,B 0,C 180,E1 -9505.323,E2 -9505.323} C_VEL
LIN {X 0,Y 432.324,Z 295.636,A -85,B 0,C 180,E1 -9508.654,E2 -9508.654} C_VEL
LIN {X 0,Y 432.378,Z 295.629,A -85,B 0,C 180,E1 -9511.37,E2 -9511.37} C_VEL
LIN {X 0,Y 432.587,Z 297.138,A -85,B 0,C 180,E1 -9513.982,E2 -9513.982} C_VEL
LIN {X 0,Y 432.629,Z 298.492,A -85,B 0,C 180,E1 -9516.039,E2 -9516.039} C_VEL
LIN {X 0,Y 432.582,Z 300.679,A -85,B 0,C 180,E1 -9519.058,E2 -9519.058} C_VEL
LIN {X 0,Y 432.445,Z 302.977,A -85,B 0,C 180,E1 -9522.014,E2 -9522.014} C_VEL
LIN {X 0,Y 432.461,Z 304.326,A -85,B 0,C 180,E1 -9523.538,E2 -9523.538} C_VEL
LIN {X 0,Y 436.028,Z 315.704,A -85,B 0,C 180,E1 -9524.149,E2 -9524.149} C_VEL
LIN {X 0,Y 436.326,Z 318.451,A -85,B 0,C 180,E1 -9524.288,E2 -9524.288} C_VEL
LIN {X 0,Y 435.925,Z 330.484,A -85,B 0,C 180,E1 -9524.932,E2 -9524.932} C_VEL
LIN {X 0,Y 435.364,Z 342.896,A -85,B 0,C 180,E1 -9525.802,E2 -9525.802} C_VEL
LIN {X 0,Y 434.82,Z 354.062,A -85,B 0,C 180,E1 -9526.803,E2 -9526.803} C_VEL
LIN {X 0,Y 434.253,Z 363.54,A -85,B 0,C 180,E1 -9527.855,E2 -9527.855} C_VEL
LIN {X 0,Y 433.704,Z 372.191,A -85,B 0,C 180,E1 -9529.024,E2 -9529.024} C_VEL
LIN {X 0,Y 433.198,Z 380.628,A -85,B 0,C 180,E1 -9530.428,E2 -9530.428} C_VEL
LIN {X 0,Y 432.739,Z 387.422,A -85,B 0,C 180,E1 -9531.854,E2 -9531.854} C_VEL
LIN {X 0,Y 432.236,Z 393.429,A -85,B 0,C 180,E1 -9533.465,E2 -9533.465} C_VEL
LIN {X 0,Y 432.098,Z 397.327,A -85,B 0,C 180,E1 -9534.868,E2 -9534.868} C_VEL
LIN {X 0,Y 431.858,Z 400.167,A -85,B 0,C 180,E1 -9536.268,E2 -9536.268} C_VEL
LIN {X 0,Y 431.635,Z 401.506,A -85,B 0,C 180,E1 -9537.2,E2 -9537.2} C_VEL
LIN {X 0,Y 431.458,Z 402.913,A -85,B 0,C 180,E1 -9539.067,E2 -9539.067} C_VEL
LIN {X 0,Y 431.434,Z 403.008,A -85,B 0,C 180,E1 -9540,E2 -9540} C_VEL
LIN {X 0,Y 431.428,Z 402.653,A -85,B 0,C 180,E1 -9540.933,E2 -9540.933} C_VEL
LIN {X 0,Y 431.474,Z 401.895,A -85,B 0,C 180,E1 -9541.867,E2 -9541.867} C_VEL
LIN {X 0,Y 431.621,Z 400.731,A -85,B 0,C 180,E1 -9542.8,E2 -9542.8} C_VEL
LIN {X 0,Y 431.888,Z 398.149,A -85,B 0,C 180,E1 -9544.199,E2 -9544.199} C_VEL
LIN {X 0,Y 431.933,Z 394.569,A -85,B 0,C 180,E1 -9545.603,E2 -9545.603} C_VEL
LIN {X 0,Y 432.182,Z 388.828,A -85,B 0,C 180,E1 -9547.268,E2 -9547.268} C_VEL
LIN {X 0,Y 432.563,Z 381.562,A -85,B 0,C 180,E1 -9548.879,E2 -9548.879} C_VEL
LIN {X 0,Y 432.978,Z 373.521,A -85,B 0,C 180,E1 -9550.285,E2 -9550.285} C_VEL
LIN {X 0,Y 433.45,Z 365.315,A -85,B 0,C 180,E1 -9551.457,E2 -9551.457} C_VEL
LIN {X 0,Y 433.968,Z 355.333,A -85,B 0,C 180,E1 -9552.629,E2 -9552.629} C_VEL
LIN {X 0,Y 434.482,Z 344.783,A -85,B 0,C 180,E1 -9553.635,E2 -9553.635} C_VEL
LIN {X 0,Y 434.874,Z 333.379,A -85,B 0,C 180,E1 -9554.507,E2 -9554.507} C_VEL
LIN {X 0,Y 435.416,Z 320.583,A -85,B 0,C 180,E1 -9555.266,E2 -9555.266} C_VEL
LIN {X 0,Y 435.323,Z 314.014,A -85,B 0,C 180,E1 -9555.584,E2 -9555.584} C_VEL
LIN {X 0,Y 432.021,Z 300.174,A -85,B 0,C 180,E1 -9556.197,E2 -9556.197} C_VEL
LIN {X 0,Y 431.686,Z 298.604,A -85,B 0,C 180,E1 -9556.261,E2 -9556.261} C_VEL
LIN {X 0,Y 431.617,Z 296.453,A -85,B 0,C 180,E1 -9558.022,E2 -9558.022} C_VEL
LIN {X 0,Y 431.731,Z 295.71,A -85,B 0,C 180,E1 -9559.236,E2 -9559.236} C_VEL
LIN {X 0,Y 432.011,Z 295.671,A -85,B 0,C 180,E1 -9561.984,E2 -9561.984} C_VEL
LIN {X 0,Y 432.282,Z 295.636,A -85,B 0,C 180,E1 -9565.006,E2 -9565.006} C_VEL
LIN {X 0,Y 432.373,Z 295.624,A -85,B 0,C 180,E1 -9568.124,E2 -9568.124} C_VEL
LIN {X 0,Y 432.324,Z 295.626,A -85,B 0,C 180,E1 -9571.346,E2 -9571.346} C_VEL
LIN {X 0,Y 432.343,Z 295.627,A -85,B 0,C 180,E1 -9574.677,E2 -9574.677} C_VEL
LIN {X 0,Y 432.34,Z 295.634,A -85,B 0,C 180,E1 -9578.15,E2 -9578.15} C_VEL
LIN {X 0,Y 432.336,Z 295.633,A -85,B 0,C 180,E1 -9581.602,E2 -9581.602} C_VEL
LIN {X 0,Y 432.34,Z 295.63,A -85,B 0,C 180,E1 -9584.347,E2 -9584.347} C_VEL
LIN {X 0,Y 432.323,Z 295.63,A -85,B 0,C 180,E1 -9587.016,E2 -9587.016} C_VEL
LIN {X 0,Y 432.336,Z 295.634,A -85,B 0,C 180,E1 -9589.821,E2 -9589.821} C_VEL
LIN {X 0,Y 432.306,Z 295.634,A -85,B 0,C 180,E1 -9593.022,E2 -9593.022} C_VEL
LIN {X 0,Y 432.239,Z 295.649,A -85,B 0,C 180,E1 -9595.313,E2 -9595.313} C_VEL
LIN {X 0,Y 432.111,Z 295.734,A -85,B 0,C 180,E1 -9596.707,E2 -9596.707} C_VEL
LIN {X 0,Y 431.83,Z 302.417,A -85,B 0,C 180,E1 -9600.774,E2 -9600.774} C_VEL
LIN {X 0,Y 431.806,Z 307.509,A -85,B 0,C 180,E1 -9603.931,E2 -9603.931} C_VEL
LIN {X 0,Y 431.737,Z 312.55,A -85,B 0,C 180,E1 -9607.003,E2 -9607.003} C_VEL
LIN {X 0,Y 431.692,Z 317.665,A -85,B 0,C 180,E1 -9610.008,E2 -9610.008} C_VEL
LIN {X 0,Y 431.673,Z 323.855,A -85,B 0,C 180,E1 -9613.394,E2 -9613.394} C_VEL
LIN {X 0,Y 434.923,Z 337.073,A -85,B 0,C 180,E1 -9613.916,E2 -9613.916} C_VEL
LIN {X 0,Y 436.141,Z 343.371,A -85,B 0,C 180,E1 -9614.221,E2 -9614.221} C_VEL
LIN {X 0,Y 435.73,Z 354.774,A -85,B 0,C 180,E1 -9614.805,E2 -9614.805} C_VEL
LIN {X 0,Y 435.205,Z 365.291,A -85,B 0,C 180,E1 -9615.505,E2 -9615.505} C_VEL
LIN {X 0,Y 434.662,Z 376.544,A -85,B 0,C 180,E1 -9616.46,E2 -9616.46} C_VEL
LIN {X 0,Y 434.085,Z 386.359,A -85,B 0,C 180,E1 -9617.494,E2 -9617.494} C_VEL
LIN {X 0,Y 433.517,Z 394.576,A -85,B 0,C 180,E1 -9618.545,E2 -9618.545} C_VEL
LIN {X 0,Y 432.881,Z 403.48,A -85,B 0,C 180,E1 -9619.949,E2 -9619.949} C_VEL
LIN {X 0,Y 432.372,Z 410.633,A -85,B 0,C 180,E1 -9621.353,E2 -9621.353} C_VEL
LIN {X 0,Y 431.984,Z 416.521,A -85,B 0,C 180,E1 -9622.806,E2 -9622.806} C_VEL
LIN {X 0,Y 431.218,Z 418.998,A -85,B 0,C 180,E1 -9623.511,E2 -9623.511} C_VEL
LIN {X 0,Y 428.205,Z 422.557,A -85,B 0,C 180,E1 -9624.677,E2 -9624.677} C_VEL
LIN {X 0,Y 425.669,Z 424.911,A -85,B 0,C 180,E1 -9625.643,E2 -9625.643} C_VEL
LIN {X 0,Y 424.54,Z 426.353,A -85,B 0,C 180,E1 -9626.405,E2 -9626.405} C_VEL
LIN {X 0,Y 424.425,Z 426.711,A -85,B 0,C 180,E1 -9626.666,E2 -9626.666} C_VEL
LIN {X 0,Y 424.286,Z 428.428,A -85,B 0,C 180,E1 -9628.102,E2 -9628.102} C_VEL
LIN {X 0,Y 424.229,Z 429.275,A -85,B 0,C 180,E1 -9630,E2 -9630} C_VEL
LIN {X 0,Y 424.287,Z 428.504,A -85,B 0,C 180,E1 -9631.898,E2 -9631.898} C_VEL
LIN {X 0,Y 424.493,Z 426.186,A -85,B 0,C 180,E1 -9633.797,E2 -9633.797} C_VEL
LIN {X 0,Y 424.47,Z 423.348,A -85,B 0,C 180,E1 -9635.225,E2 -9635.225} C_VEL
LIN {X 0,Y 424.87,Z 419.467,A -85,B 0,C 180,E1 -9636.649,E2 -9636.649} C_VEL
LIN {X 0,Y 425.099,Z 414.46,A -85,B 0,C 180,E1 -9638.078,E2 -9638.078} C_VEL
LIN {X 0,Y 425.572,Z 408.128,A -85,B 0,C 180,E1 -9639.506,E2 -9639.506} C_VEL
LIN {X 0,Y 426.155,Z 400.258,A -85,B 0,C 180,E1 -9640.933,E2 -9640.933} C_VEL
LIN {X 0,Y 426.749,Z 392.216,A -85,B 0,C 180,E1 -9642.121,E2 -9642.121} C_VEL
LIN {X 0,Y 427.458,Z 382.349,A -85,B 0,C 180,E1 -9643.308,E2 -9643.308} C_VEL
LIN {X 0,Y 428.021,Z 371.499,A -85,B 0,C 180,E1 -9644.357,E2 -9644.357} C_VEL
LIN {X 0,Y 428.716,Z 360.354,A -85,B 0,C 180,E1 -9645.206,E2 -9645.206} C_VEL
LIN {X 0,Y 429.2,Z 348.176,A -85,B 0,C 180,E1 -9645.919,E2 -9645.919} C_VEL
LIN {X 0,Y 429.07,Z 343.138,A -85,B 0,C 180,E1 -9646.168,E2 -9646.168} C_VEL
LIN {X 0,Y 426.49,Z 331.348,A -85,B 0,C 180,E1 -9646.717,E2 -9646.717} C_VEL
LIN {X 0,Y 424.632,Z 324.17,A -85,B 0,C 180,E1 -9647.012,E2 -9647.012} C_VEL
LIN {X 0,Y 424.635,Z 318.111,A -85,B 0,C 180,E1 -9650.339,E2 -9650.339} C_VEL
LIN {X 0,Y 424.698,Z 312.908,A -85,B 0,C 180,E1 -9653.401,E2 -9653.401} C_VEL
LIN {X 0,Y 424.767,Z 307.559,A -85,B 0,C 180,E1 -9656.688,E2 -9656.688} C_VEL
LIN {X 0,Y 424.797,Z 302.602,A -85,B 0,C 180,E1 -9659.758,E2 -9659.758} C_VEL
LIN {X 0,Y 425.084,Z 296.541,A -85,B 0,C 180,E1 -9663.49,E2 -9663.49} C_VEL
LIN {X 0,Y 425.262,Z 296.516,A -85,B 0,C 180,E1 -9665.924,E2 -9665.924} C_VEL
LIN {X 0,Y 425.296,Z 296.51,A -85,B 0,C 180,E1 -9669.043,E2 -9669.043} C_VEL
LIN {X 0,Y 425.277,Z 296.515,A -85,B 0,C 180,E1 -9672.653,E2 -9672.653} C_VEL
LIN {X 0,Y 425.264,Z 296.514,A -85,B 0,C 180,E1 -9676.044,E2 -9676.044} C_VEL
LIN {X 0,Y 425.278,Z 296.511,A -85,B 0,C 180,E1 -9678.621,E2 -9678.621} C_VEL
LIN {X 0,Y 425.315,Z 296.507,A -85,B 0,C 180,E1 -9681.103,E2 -9681.103} C_VEL
LIN {X 0,Y 425.22,Z 296.516,A -85,B 0,C 180,E1 -9684.656,E2 -9684.656} C_VEL
LIN {X 0,Y 424.978,Z 296.609,A -85,B 0,C 180,E1 -9687.019,E2 -9687.019} C_VEL
LIN {X 0,Y 424.797,Z 302.033,A -85,B 0,C 180,E1 -9690.242,E2 -9690.242} C_VEL
LIN {X 0,Y 424.703,Z 307.405,A -85,B 0,C 180,E1 -9693.461,E2 -9693.461} C_VEL
LIN {X 0,Y 424.674,Z 312.639,A -85,B 0,C 180,E1 -9696.598,E2 -9696.598} C_VEL
LIN {X 0,Y 424.605,Z 317.768,A -85,B 0,C 180,E1 -9699.66,E2 -9699.66} C_VEL
LIN {X 0,Y 424.571,Z 321.139,A -85,B 0,C 180,E1 -9701.669,E2 -9701.669} C_VEL
LIN {X 0,Y 424.594,Z 324.366,A -85,B 0,C 180,E1 -9703.607,E2 -9703.607} C_VEL
LIN {X 0,Y 427.497,Z 338.274,A -85,B 0,C 180,E1 -9704.181,E2 -9704.181} C_VEL
LIN {X 0,Y 428.363,Z 344.609,A -85,B 0,C 180,E1 -9704.497,E2 -9704.497} C_VEL
LIN {X 0,Y 427.855,Z 356.072,A -85,B 0,C 180,E1 -9705.128,E2 -9705.128} C_VEL
LIN {X 0,Y 427.383,Z 366.795,A -85,B 0,C 180,E1 -9705.884,E2 -9705.884} C_VEL
LIN {X 0,Y 426.912,Z 378.399,A -85,B 0,C 180,E1 -9706.917,E2 -9706.917} C_VEL
LIN {X 0,Y 426.388,Z 387.19,A -85,B 0,C 180,E1 -9707.869,E2 -9707.869} C_VEL
LIN {X 0,Y 425.878,Z 396.313,A -85,B 0,C 180,E1 -9709.06,E2 -9709.06} C_VEL
LIN {X 0,Y 425.375,Z 405.151,A -85,B 0,C 180,E1 -9710.49,E2 -9710.49} C_VEL
LIN {X 0,Y 424.983,Z 412.294,A -85,B 0,C 180,E1 -9711.919,E2 -9711.919} C_VEL
LIN {X 0,Y 424.718,Z 417.955,A -85,B 0,C 180,E1 -9713.348,E2 -9713.348} C_VEL
LIN {X 0,Y 424.452,Z 422.391,A -85,B 0,C 180,E1 -9714.775,E2 -9714.775} C_VEL
LIN {X 0,Y 424.499,Z 425.707,A -85,B 0,C 180,E1 -9716.203,E2 -9716.203} C_VEL
LIN {X 0,Y 424.378,Z 427.365,A -85,B 0,C 180,E1 -9717.152,E2 -9717.152} C_VEL
LIN {X 0,Y 424.287,Z 428.584,A -85,B 0,C 180,E1 -9718.101,E2 -9718.101} C_VEL
LIN {X 0,Y 424.259,Z 429.349,A -85,B 0,C 180,E1 -9719.051,E2 -9719.051} C_VEL
LIN {X 0,Y 424.232,Z 429.72,A -85,B 0,C 180,E1 -9720,E2 -9720} C_VEL
LIN {X 0,Y 424.261,Z 429.673,A -85,B 0,C 180,E1 -9720.949,E2 -9720.949} C_VEL
LIN {X 0,Y 424.367,Z 429.167,A -85,B 0,C 180,E1 -9721.898,E2 -9721.898} C_VEL
LIN {X 0,Y 424.448,Z 428.267,A -85,B 0,C 180,E1 -9722.847,E2 -9722.847} C_VEL
LIN {X 0,Y 424.518,Z 426.949,A -85,B 0,C 180,E1 -9723.797,E2 -9723.797} C_VEL
LIN {X 0,Y 424.614,Z 424.108,A -85,B 0,C 180,E1 -9725.223,E2 -9725.223} C_VEL
LIN {X 0,Y 424.89,Z 420.168,A -85,B 0,C 180,E1 -9726.649,E2 -9726.649} C_VEL
LIN {X 0,Y 425.176,Z 415.032,A -85,B 0,C 180,E1 -9728.077,E2 -9728.077} C_VEL
LIN {X 0,Y 425.635,Z 408.535,A -85,B 0,C 180,E1 -9729.504,E2 -9729.504} C_VEL
LIN {X 0,Y 426.167,Z 400.421,A -85,B 0,C 180,E1 -9730.932,E2 -9730.932} C_VEL
LIN {X 0,Y 426.684,Z 392.079,A -85,B 0,C 180,E1 -9732.123,E2 -9732.123} C_VEL
LIN {X 0,Y 427.348,Z 381.895,A -85,B 0,C 180,E1 -9733.311,E2 -9733.311} C_VEL
LIN {X 0,Y 427.932,Z 371.225,A -85,B 0,C 180,E1 -9734.311,E2 -9734.311} C_VEL
LIN {X 0,Y 428.576,Z 359.154,A -85,B 0,C 180,E1 -9735.211,E2 -9735.211} C_VEL
LIN {X 0,Y 429.177,Z 345.566,A -85,B 0,C 180,E1 -9735.981,E2 -9735.981} C_VEL
LIN {X 0,Y 428.764,Z 341.81,A -85,B 0,C 180,E1 -9736.18,E2 -9736.18} C_VEL
LIN {X 0,Y 425.77,Z 330.109,A -85,B 0,C 180,E1 -9736.787,E2 -9736.787} C_VEL
LIN {X 0,Y 424.969,Z 327.35,A -85,B 0,C 180,E1 -9736.917,E2 -9736.917} C_VEL
LIN {X 0,Y 425.033,Z 321.418,A -85,B 0,C 180,E1 -9740.319,E2 -9740.319} C_VEL
LIN {X 0,Y 425.05,Z 315.93,A -85,B 0,C 180,E1 -9743.38,E2 -9743.38} C_VEL
LIN {X 0,Y 425.075,Z 310.114,A -85,B 0,C 180,E1 -9746.513,E2 -9746.513} C_VEL
LIN {X 0,Y 425.219,Z 303.777,A -85,B 0,C 180,E1 -9749.725,E2 -9749.725} C_VEL
LIN {X 0,Y 425.243,Z 297.854,A -85,B 0,C 180,E1 -9752.554,E2 -9752.554} C_VEL
LIN {X 0,Y 425.159,Z 296.529,A -85,B 0,C 180,E1 -9753.271,E2 -9753.271} C_VEL
LIN {X 0,Y 425.272,Z 296.514,A -85,B 0,C 180,E1 -9755.926,E2 -9755.926} C_VEL
LIN {X 0,Y 425.284,Z 296.513,A -85,B 0,C 180,E1 -9759.041,E2 -9759.041} C_VEL
LIN {X 0,Y 425.284,Z 296.511,A -85,B 0,C 180,E1 -9761.957,E2 -9761.957} C_VEL
LIN {X 0,Y 425.287,Z 296.509,A -85,B 0,C 180,E1 -9765.283,E2 -9765.283} C_VEL
LIN {X 0,Y 425.307,Z 296.634,A -85,B 0,C 180,E1 -9766.302,E2 -9766.302} C_VEL
LIN {X 0,Y 426.687,Z 303.567,A -85,B 0,C 180,E1 -9769.259,E2 -9769.259} C_VEL
LIN {X 0,Y 427.955,Z 310.349,A -85,B 0,C 180,E1 -9772.024,E2 -9772.024} C_VEL
LIN {X 0,Y 428.471,Z 314.946,A -85,B 0,C 180,E1 -9773.808,E2 -9773.808} C_VEL
LIN {X 0,Y 427.776,Z 323.528,A -85,B 0,C 180,E1 -9776.918,E2 -9776.918} C_VEL
LIN {X 0,Y 427.08,Z 333.482,A -85,B 0,C 180,E1 -9780.417,E2 -9780.417} C_VEL
LIN {X 0,Y 426.353,Z 344.298,A -85,B 0,C 180,E1 -9784.098,E2 -9784.098} C_VEL
LIN {X 0,Y 425.932,Z 352.014,A -85,B 0,C 180,E1 -9786.671,E2 -9786.671} C_VEL
LIN {X 0,Y 425.475,Z 361.33,A -85,B 0,C 180,E1 -9789.703,E2 -9789.703} C_VEL
LIN {X 0,Y 425.05,Z 371.427,A -85,B 0,C 180,E1 -9792.95,E2 -9792.95} C_VEL
LIN {X 0,Y 427.285,Z 386.786,A -85,B 0,C 180,E1 -9793.523,E2 -9793.523} C_VEL
LIN {X 0,Y 428.732,Z 397.451,A -85,B 0,C 180,E1 -9794.063,E2 -9794.063} C_VEL
LIN {X 0,Y 428.077,Z 409.49,A -85,B 0,C 180,E1 -9794.771,E2 -9794.771} C_VEL
LIN {X 0,Y 427.283,Z 421.846,A -85,B 0,C 180,E1 -9795.716,E2 -9795.716} C_VEL
LIN {X 0,Y 426.634,Z 432.836,A -85,B 0,C 180,E1 -9796.787,E2 -9796.787} C_VEL
LIN {X 0,Y 425.913,Z 443.573,A -85,B 0,C 180,E1 -9798.097,E2 -9798.097} C_VEL
LIN {X 0,Y 425.359,Z 451.535,A -85,B 0,C 180,E1 -9799.288,E2 -9799.288} C_VEL
LIN {X 0,Y 424.898,Z 459.355,A -85,B 0,C 180,E1 -9800.719,E2 -9800.719} C_VEL
LIN {X 0,Y 424.582,Z 464.69,A -85,B 0,C 180,E1 -9801.912,E2 -9801.912} C_VEL
LIN {X 0,Y 424.377,Z 470.487,A -85,B 0,C 180,E1 -9803.539,E2 -9803.539} C_VEL
LIN {X 0,Y 424.228,Z 474.997,A -85,B 0,C 180,E1 -9805.249,E2 -9805.249} C_VEL
LIN {X 0,Y 424.159,Z 476.881,A -85,B 0,C 180,E1 -9806.2,E2 -9806.2} C_VEL
LIN {X 0,Y 424.216,Z 478.305,A -85,B 0,C 180,E1 -9807.151,E2 -9807.151} C_VEL
LIN {X 0,Y 424.185,Z 479.302,A -85,B 0,C 180,E1 -9808.101,E2 -9808.101} C_VEL
LIN {X 0,Y 424.204,Z 479.9,A -85,B 0,C 180,E1 -9809.051,E2 -9809.051} C_VEL
LIN {X 0,Y 424.177,Z 480.094,A -85,B 0,C 180,E1 -9810,E2 -9810} C_VEL
LIN {X 0,Y 424.205,Z 479.852,A -85,B 0,C 180,E1 -9810.949,E2 -9810.949} C_VEL
LIN {X 0,Y 424.212,Z 479.2,A -85,B 0,C 180,E1 -9811.899,E2 -9811.899} C_VEL
LIN {X 0,Y 424.218,Z 478.141,A -85,B 0,C 180,E1 -9812.849,E2 -9812.849} C_VEL
LIN {X 0,Y 424.178,Z 476.664,A -85,B 0,C 180,E1 -9813.8,E2 -9813.8} C_VEL
LIN {X 0,Y 424.321,Z 473.601,A -85,B 0,C 180,E1 -9815.227,E2 -9815.227} C_VEL
LIN {X 0,Y 424.399,Z 469.457,A -85,B 0,C 180,E1 -9816.657,E2 -9816.657} C_VEL
LIN {X 0,Y 424.666,Z 463.111,A -85,B 0,C 180,E1 -9818.326,E2 -9818.326} C_VEL
LIN {X 0,Y 425.027,Z 456.197,A -85,B 0,C 180,E1 -9819.758,E2 -9819.758} C_VEL
LIN {X 0,Y 425.543,Z 447.652,A -85,B 0,C 180,E1 -9821.19,E2 -9821.19} C_VEL
LIN {X 0,Y 426.073,Z 438.894,A -85,B 0,C 180,E1 -9822.382,E2 -9822.382} C_VEL
LIN {X 0,Y 426.771,Z 428.647,A -85,B 0,C 180,E1 -9823.524,E2 -9823.524} C_VEL
LIN {X 0,Y 427.354,Z 417.644,A -85,B 0,C 180,E1 -9824.524,E2 -9824.524} C_VEL
LIN {X 0,Y 428.105,Z 406.229,A -85,B 0,C 180,E1 -9825.35,E2 -9825.35} C_VEL
LIN {X 0,Y 428.489,Z 395.902,A -85,B 0,C 180,E1 -9825.946,E2 -9825.946} C_VEL
LIN {X 0,Y 426.543,Z 381.716,A -85,B 0,C 180,E1 -9826.641,E2 -9826.641} C_VEL
LIN {X 0,Y 424.991,Z 369.288,A -85,B 0,C 180,E1 -9827.106,E2 -9827.106} C_VEL
LIN {X 0,Y 425.298,Z 358.967,A -85,B 0,C 180,E1 -9830.305,E2 -9830.305} C_VEL
LIN {X 0,Y 425.716,Z 349.352,A -85,B 0,C 180,E1 -9833.341,E2 -9833.341} C_VEL
LIN {X 0,Y 426.146,Z 339.858,A -85,B 0,C 180,E1 -9836.442,E2 -9836.442} C_VEL
LIN {X 0,Y 426.774,Z 329.034,A -85,B 0,C 180,E1 -9840.15,E2 -9840.15} C_VEL
LIN {X 0,Y 427.464,Z 320.142,A -85,B 0,C 180,E1 -9843.428,E2 -9843.428} C_VEL
LIN {X 0,Y 428.142,Z 313.225,A -85,B 0,C 180,E1 -9846.224,E2 -9846.224} C_VEL
LIN {X 0,Y 427.778,Z 309.523,A -85,B 0,C 180,E1 -9847.945,E2 -9847.945} C_VEL
LIN {X 0,Y 426.841,Z 304.34,A -85,B 0,C 180,E1 -9850.765,E2 -9850.765} C_VEL
LIN {X 0,Y 425.968,Z 299.9,A -85,B 0,C 180,E1 -9853.865,E2 -9853.865} C_VEL
LIN {X 0,Y 425.39,Z 297.109,A -85,B 0,C 180,E1 -9856.631,E2 -9856.631} C_VEL
LIN {X 0,Y 425.284,Z 296.513,A -85,B 0,C 180,E1 -9857.737,E2 -9857.737} C_VEL
LIN {X 0,Y 425.299,Z 296.511,A -85,B 0,C 180,E1 -9861.101,E2 -9861.101} C_VEL
LIN {X 0,Y 425.302,Z 296.51,A -85,B 0,C 180,E1 -9864.664,E2 -9864.664} C_VEL
LIN {X 0,Y 425.268,Z 296.514,A -85,B 0,C 180,E1 -9868.073,E2 -9868.073} C_VEL
LIN {X 0,Y 425.294,Z 296.536,A -85,B 0,C 180,E1 -9870.281,E2 -9870.281} C_VEL
LIN {X 0,Y 425.598,Z 298.261,A -85,B 0,C 180,E1 -9873.522,E2 -9873.522} C_VEL
LIN {X 0,Y 425.67,Z 299.562,A -85,B 0,C 180,E1 -9875.622,E2 -9875.622} C_VEL
LIN {X 0,Y 425.604,Z 301.698,A -85,B 0,C 180,E1 -9878.698,E2 -9878.698} C_VEL
LIN {X 0,Y 425.47,Z 303.968,A -85,B 0,C 180,E1 -9881.709,E2 -9881.709} C_VEL
LIN {X 0,Y 425.446,Z 305.24,A -85,B 0,C 180,E1 -9883.204,E2 -9883.204} C_VEL
LIN {X 0,Y 429.136,Z 316.457,A -85,B 0,C 180,E1 -9883.835,E2 -9883.835} C_VEL
LIN {X 0,Y 429.613,Z 320.201,A -85,B 0,C 180,E1 -9884.036,E2 -9884.036} C_VEL
LIN {X 0,Y 429.086,Z 333.7,A -85,B 0,C 180,E1 -9884.807,E2 -9884.807} C_VEL
LIN {X 0,Y 428.552,Z 345.066,A -85,B 0,C 180,E1 -9885.653,E2 -9885.653} C_VEL
LIN {X 0,Y 427.871,Z 356.296,A -85,B 0,C 180,E1 -9886.705,E2 -9886.705} C_VEL
LIN {X 0,Y 427.288,Z 366.48,A -85,B 0,C 180,E1 -9887.895,E2 -9887.895} C_VEL
LIN {X 0,Y 426.735,Z 374.73,A -85,B 0,C 180,E1 -9889.082,E2 -9889.082} C_VEL
LIN {X 0,Y 426.104,Z 382.761,A -85,B 0,C 180,E1 -9890.506,E2 -9890.506} C_VEL
LIN {X 0,Y 425.729,Z 389.367,A -85,B 0,C 180,E1 -9891.981,E2 -9891.981} C_VEL
LIN {X 0,Y 425.234,Z 394.275,A -85,B 0,C 180,E1 -9893.357,E2 -9893.357} C_VEL
LIN {X 0,Y 425.08,Z 398.148,A -85,B 0,C 180,E1 -9894.783,E2 -9894.783} C_VEL
LIN {X 0,Y 424.828,Z 400.962,A -85,B 0,C 180,E1 -9896.206,E2 -9896.206} C_VEL
LIN {X 0,Y 424.592,Z 402.276,A -85,B 0,C 180,E1 -9897.154,E2 -9897.154} C_VEL
LIN {X 0,Y 424.454,Z 403.164,A -85,B 0,C 180,E1 -9898.102,E2 -9898.102} C_VEL
LIN {X 0,Y 424.397,Z 403.645,A -85,B 0,C 180,E1 -9899.051,E2 -9899.051} C_VEL
LIN {X 0,Y 424.369,Z 403.707,A -85,B 0,C 180,E1 -9900,E2 -9900} C_VEL
LIN {X 0,Y 424.365,Z 403.326,A -85,B 0,C 180,E1 -9900.949,E2 -9900.949} C_VEL
LIN {X 0,Y 424.42,Z 402.545,A -85,B 0,C 180,E1 -9901.898,E2 -9901.898} C_VEL
LIN {X 0,Y 424.579,Z 401.356,A -85,B 0,C 180,E1 -9902.846,E2 -9902.846} C_VEL
LIN {X 0,Y 424.852,Z 398.733,A -85,B 0,C 180,E1 -9904.269,E2 -9904.269} C_VEL
LIN {X 0,Y 424.876,Z 395.108,A -85,B 0,C 180,E1 -9905.696,E2 -9905.696} C_VEL
LIN {X 0,Y 425.154,Z 389.53,A -85,B 0,C 180,E1 -9907.327,E2 -9907.327} C_VEL
LIN {X 0,Y 425.477,Z 383.117,A -85,B 0,C 180,E1 -9908.789,E2 -9908.789} C_VEL
LIN {X 0,Y 425.939,Z 375.317,A -85,B 0,C 180,E1 -9910.217,E2 -9910.217} C_VEL
LIN {X 0,Y 426.383,Z 367.345,A -85,B 0,C 180,E1 -9911.408,E2 -9911.408} C_VEL
LIN {X 0,Y 426.964,Z 356.539,A -85,B 0,C 180,E1 -9912.718,E2 -9912.718} C_VEL
LIN {X 0,Y 427.541,Z 345.402,A -85,B 0,C 180,E1 -9913.804,E2 -9913.804} C_VEL
LIN {X 0,Y 427.972,Z 333.199,A -85,B 0,C 180,E1 -9914.746,E2 -9914.746} C_VEL
LIN {X 0,Y 428.537,Z 320.527,A -85,B 0,C 180,E1 -9915.498,E2 -9915.498} C_VEL
LIN {X 0,Y 428.535,Z 315.735,A -85,B 0,C 180,E1 -9915.735,E2 -9915.735} C_VEL
LIN {X 0,Y 425.355,Z 302.247,A -85,B 0,C 180,E1 -9916.362,E2 -9916.362} C_VEL
LIN {X 0,Y 424.633,Z 299.101,A -85,B 0,C 180,E1 -9916.514,E2 -9916.514} C_VEL
LIN {X 0,Y 424.562,Z 296.905,A -85,B 0,C 180,E1 -9918.332,E2 -9918.332} C_VEL
LIN {X 0,Y 424.783,Z 296.573,A -85,B 0,C 180,E1 -9920.331,E2 -9920.331} C_VEL
LIN {X 0,Y 425.099,Z 296.534,A -85,B 0,C 180,E1 -9923.377,E2 -9923.377} C_VEL
LIN {X 0,Y 425.239,Z 296.51,A -85,B 0,C 180,E1 -9925.449,E2 -9925.449} C_VEL
LIN {X 0,Y 425.334,Z 296.507,A -85,B 0,C 180,E1 -9928.632,E2 -9928.632} C_VEL
LIN {X 0,Y 425.267,Z 296.507,A -85,B 0,C 180,E1 -9931.927,E2 -9931.927} C_VEL
LIN {X 0,Y 425.302,Z 296.501,A -85,B 0,C 180,E1 -9935.336,E2 -9935.336} C_VEL
LIN {X 0,Y 425.296,Z 296.506,A -85,B 0,C 180,E1 -9939.043,E2 -9939.043} C_VEL
LIN {X 0,Y 425.278,Z 296.511,A -85,B 0,C 180,E1 -9942.653,E2 -9942.653} C_VEL
LIN {X 0,Y 425.264,Z 296.513,A -85,B 0,C 180,E1 -9946.044,E2 -9946.044} C_VEL
LIN {X 0,Y 425.277,Z 296.508,A -85,B 0,C 180,E1 -9948.621,E2 -9948.621} C_VEL
LIN {X 0,Y 425.309,Z 296.507,A -85,B 0,C 180,E1 -9951.102,E2 -9951.102} C_VEL
LIN {X 0,Y 425.253,Z 296.516,A -85,B 0,C 180,E1 -9954.659,E2 -9954.659} C_VEL
LIN {X 0,Y 425.063,Z 296.551,A -85,B 0,C 180,E1 -9956.65,E2 -9956.65} C_VEL
LIN {X 0,Y 424.796,Z 302.439,A -85,B 0,C 180,E1 -9960.242,E2 -9960.242} C_VEL
LIN {X 0,Y 424.774,Z 307.618,A -85,B 0,C 180,E1 -9963.466,E2 -9963.466} C_VEL
LIN {X 0,Y 424.697,Z 312.743,A -85,B 0,C 180,E1 -9966.599,E2 -9966.599} C_VEL
LIN {X 0,Y 424.635,Z 317.935,A -85,B 0,C 180,E1 -9969.661,E2 -9969.661} C_VEL
LIN {X 0,Y 424.626,Z 324.211,A -85,B 0,C 180,E1 -9973.108,E2 -9973.108} C_VEL
LIN {X 0,Y 427.929,Z 337.629,A -85,B 0,C 180,E1 -9973.652,E2 -9973.652} C_VEL
LIN {X 0,Y 429.272,Z 345.049,A -85,B 0,C 180,E1 -9974.023,E2 -9974.023} C_VEL
LIN {X 0,Y 428.819,Z 357.066,A -85,B 0,C 180,E1 -9974.676,E2 -9974.676} C_VEL
LIN {X 0,Y 428.276,Z 367.639,A -85,B 0,C 180,E1 -9975.421,E2 -9975.421} C_VEL
LIN {X 0,Y 427.71,Z 378.324,A -85,B 0,C 180,E1 -9976.369,E2 -9976.369} C_VEL
LIN {X 0,Y 427.109,Z 387.761,A -85,B 0,C 180,E1 -9977.407,E2 -9977.407} C_VEL
LIN {X 0,Y 426.433,Z 396.596,A -85,B 0,C 180,E1 -9978.593,E2 -9978.593} C_VEL
LIN {X 0,Y 425.809,Z 405.209,A -85,B 0,C 180,E1 -9980.02,E2 -9980.02} C_VEL
LIN {X 0,Y 425.274,Z 412.116,A -85,B 0,C 180,E1 -9981.446,E2 -9981.446} C_VEL
LIN {X 0,Y 424.911,Z 417.793,A -85,B 0,C 180,E1 -9982.932,E2 -9982.932} C_VEL
LIN {X 0,Y 424.564,Z 421.915,A -85,B 0,C 180,E1 -9984.3,E2 -9984.3} C_VEL
LIN {X 0,Y 424.523,Z 424.177,A -85,B 0,C 180,E1 -9985.252,E2 -9985.252} C_VEL
LIN {X 0,Y 424.425,Z 426.711,A -85,B 0,C 180,E1 -9986.666,E2 -9986.666} C_VEL
LIN {X 0,Y 423.67,Z 427.833,A -85,B 0,C 180,E1 -9987.444,E2 -9987.444} C_VEL
LIN {X 0,Y 420.696,Z 429.088,A -85,B 0,C 180,E1 -9988.716,E2 -9988.716} C_VEL
LIN {X 0,Y 418.237,Z 429.586,A -85,B 0,C 180,E1 -9989.749,E2 -9989.749} C_VEL
LIN {X 0,Y 417.207,Z 429.613,A -85,B 0,C 180,E1 -9990.551,E2 -9990.551} C_VEL
LIN {X 0,Y 417.135,Z 429.529,A -85,B 0,C 180,E1 -9990.822,E2 -9990.822} C_VEL
LIN {X 0,Y 417.209,Z 428.918,A -85,B 0,C 180,E1 -9991.931,E2 -9991.931} C_VEL
LIN {X 0,Y 417.435,Z 426.599,A -85,B 0,C 180,E1 -9993.862,E2 -9993.862} C_VEL
LIN {X 0,Y 417.413,Z 423.761,A -85,B 0,C 180,E1 -9995.313,E2 -9995.313} C_VEL
LIN {X 0,Y 417.817,Z 419.88,A -85,B 0,C 180,E1 -9996.762,E2 -9996.762} C_VEL
LIN {X 0,Y 418.089,Z 414.87,A -85,B 0,C 180,E1 -9998.215,E2 -9998.215} C_VEL
LIN {X 0,Y 418.596,Z 408.536,A -85,B 0,C 180,E1 -9999.665,E2 -9999.665} C_VEL
LIN {X 0,Y 419.182,Z 400.666,A -85,B 0,C 180,E1 -10001.117,E2 -10001.117} C_VEL
LIN {X 0,Y 419.82,Z 392.62,A -85,B 0,C 180,E1 -10002.324,E2 -10002.324} C_VEL
LIN {X 0,Y 420.577,Z 382.748,A -85,B 0,C 180,E1 -10003.53,E2 -10003.53} C_VEL
LIN {X 0,Y 421.186,Z 371.77,A -85,B 0,C 180,E1 -10004.606,E2 -10004.606} C_VEL
LIN {X 0,Y 421.902,Z 360.74,A -85,B 0,C 180,E1 -10005.458,E2 -10005.458} C_VEL
LIN {X 0,Y 422.393,Z 348.547,A -85,B 0,C 180,E1 -10006.182,E2 -10006.182} C_VEL
LIN {X 0,Y 422.25,Z 344.316,A -85,B 0,C 180,E1 -10006.401,E2 -10006.401} C_VEL
LIN {X 0,Y 419.672,Z 332.53,A -85,B 0,C 180,E1 -10006.971,E2 -10006.971} C_VEL
LIN {X 0,Y 417.597,Z 324.527,A -85,B 0,C 180,E1 -10007.307,E2 -10007.307} C_VEL
LIN {X 0,Y 417.598,Z 318.376,A -85,B 0,C 180,E1 -10010.697,E2 -10010.697} C_VEL
LIN {X 0,Y 417.651,Z 314.861,A -85,B 0,C 180,E1 -10012.77,E2 -10012.77} C_VEL
LIN {X 0,Y 417.682,Z 309.631,A -85,B 0,C 180,E1 -10015.943,E2 -10015.943} C_VEL
LIN {X 0,Y 417.751,Z 304.407,A -85,B 0,C 180,E1 -10019.201,E2 -10019.201} C_VEL
LIN {X 0,Y 418.048,Z 297.527,A -85,B 0,C 180,E1 -10023.441,E2 -10023.441} C_VEL
LIN {X 0,Y 418.231,Z 297.391,A -85,B 0,C 180,E1 -10026.235,E2 -10026.235} C_VEL
LIN {X 0,Y 418.251,Z 297.389,A -85,B 0,C 180,E1 -10029.682,E2 -10029.682} C_VEL
LIN {X 0,Y 418.232,Z 297.392,A -85,B 0,C 180,E1 -10032.321,E2 -10032.321} C_VEL
LIN {X 0,Y 418.238,Z 297.391,A -85,B 0,C 180,E1 -10035.109,E2 -10035.109} C_VEL
LIN {X 0,Y 418.242,Z 297.389,A -85,B 0,C 180,E1 -10037.767,E2 -10037.767} C_VEL
LIN {X 0,Y 418.261,Z 297.385,A -85,B 0,C 180,E1 -10040.618,E2 -10040.618} C_VEL
LIN {X 0,Y 418.195,Z 297.396,A -85,B 0,C 180,E1 -10043.971,E2 -10043.971} C_VEL
LIN {X 0,Y 417.928,Z 297.478,A -85,B 0,C 180,E1 -10047.035,E2 -10047.035} C_VEL
LIN {X 0,Y 417.718,Z 303.764,A -85,B 0,C 180,E1 -10050.796,E2 -10050.796} C_VEL
LIN {X 0,Y 417.631,Z 309.187,A -85,B 0,C 180,E1 -10054.053,E2 -10054.053} C_VEL
LIN {X 0,Y 417.599,Z 314.448,A -85,B 0,C 180,E1 -10057.227,E2 -10057.227} C_VEL
LIN {X 0,Y 417.585,Z 319.834,A -85,B 0,C 180,E1 -10060.474,E2 -10060.474} C_VEL
LIN {X 0,Y 417.535,Z 324.779,A -85,B 0,C 180,E1 -10063.389,E2 -10063.389} C_VEL
LIN {X 0,Y 420.346,Z 338.129,A -85,B 0,C 180,E1 -10063.941,E2 -10063.941} C_VEL
LIN {X 0,Y 421.377,Z 343.9,A -85,B 0,C 180,E1 -10064.236,E2 -10064.236} C_VEL
LIN {X 0,Y 420.966,Z 355.533,A -85,B 0,C 180,E1 -10064.879,E2 -10064.879} C_VEL
LIN {X 0,Y 420.44,Z 367.04,A -85,B 0,C 180,E1 -10065.694,E2 -10065.694} C_VEL
LIN {X 0,Y 419.974,Z 378.202,A -85,B 0,C 180,E1 -10066.697,E2 -10066.697} C_VEL
LIN {X 0,Y 419.282,Z 389.1,A -85,B 0,C 180,E1 -10067.905,E2 -10067.905} C_VEL
LIN {X 0,Y 418.795,Z 397.923,A -85,B 0,C 180,E1 -10069.118,E2 -10069.118} C_VEL
LIN {X 0,Y 418.267,Z 406.581,A -85,B 0,C 180,E1 -10070.571,E2 -10070.571} C_VEL
LIN {X 0,Y 417.888,Z 413.491,A -85,B 0,C 180,E1 -10072.025,E2 -10072.025} C_VEL
LIN {X 0,Y 417.624,Z 419.829,A -85,B 0,C 180,E1 -10073.72,E2 -10073.72} C_VEL
LIN {X 0,Y 417.376,Z 423.945,A -85,B 0,C 180,E1 -10075.17,E2 -10075.17} C_VEL
LIN {X 0,Y 417.428,Z 426.045,A -85,B 0,C 180,E1 -10076.138,E2 -10076.138} C_VEL
LIN {X 0,Y 417.313,Z 427.726,A -85,B 0,C 180,E1 -10077.104,E2 -10077.104} C_VEL
LIN {X 0,Y 417.21,Z 428.986,A -85,B 0,C 180,E1 -10078.069,E2 -10078.069} C_VEL
LIN {X 0,Y 417.173,Z 429.775,A -85,B 0,C 180,E1 -10079.035,E2 -10079.035} C_VEL
LIN {X 0,Y 417.174,Z 430.167,A -85,B 0,C 180,E1 -10080,E2 -10080} C_VEL
LIN {X 0,Y 417.206,Z 430.149,A -85,B 0,C 180,E1 -10080.965,E2 -10080.965} C_VEL
LIN {X 0,Y 417.299,Z 429.664,A -85,B 0,C 180,E1 -10081.93,E2 -10081.93} C_VEL
LIN {X 0,Y 417.377,Z 428.78,A -85,B 0,C 180,E1 -10082.896,E2 -10082.896} C_VEL
LIN {X 0,Y 417.467,Z 427.482,A -85,B 0,C 180,E1 -10083.861,E2 -10083.861} C_VEL
LIN {X 0,Y 417.554,Z 424.665,A -85,B 0,C 180,E1 -10085.312,E2 -10085.312} C_VEL
LIN {X 0,Y 417.863,Z 420.753,A -85,B 0,C 180,E1 -10086.761,E2 -10086.761} C_VEL
LIN {X 0,Y 418.179,Z 415.66,A -85,B 0,C 180,E1 -10088.213,E2 -10088.213} C_VEL
LIN {X 0,Y 418.679,Z 409.21,A -85,B 0,C 180,E1 -10089.663,E2 -10089.663} C_VEL
LIN {X 0,Y 419.239,Z 401.133,A -85,B 0,C 180,E1 -10091.115,E2 -10091.115} C_VEL
LIN {X 0,Y 419.863,Z 390.979,A -85,B 0,C 180,E1 -10092.568,E2 -10092.568} C_VEL
LIN {X 0,Y 420.62,Z 381.024,A -85,B 0,C 180,E1 -10093.705,E2 -10093.705} C_VEL
LIN {X 0,Y 421.213,Z 370.21,A -85,B 0,C 180,E1 -10094.716,E2 -10094.716} C_VEL
LIN {X 0,Y 421.856,Z 358.471,A -85,B 0,C 180,E1 -10095.583,E2 -10095.583} C_VEL
LIN {X 0,Y 422.491,Z 345.787,A -85,B 0,C 180,E1 -10096.303,E2 -10096.303} C_VEL
LIN {X 0,Y 420.173,Z 335.415,A -85,B 0,C 180,E1 -10096.887,E2 -10096.887} C_VEL
LIN {X 0,Y 417.962,Z 327.914,A -85,B 0,C 180,E1 -10097.277,E2 -10097.277} C_VEL
LIN {X 0,Y 418.036,Z 323.725,A -85,B 0,C 180,E1 -10099.7,E2 -10099.7} C_VEL
LIN {X 0,Y 418.059,Z 318.369,A -85,B 0,C 180,E1 -10102.746,E2 -10102.746} C_VEL
LIN {X 0,Y 418.087,Z 312.576,A -85,B 0,C 180,E1 -10105.916,E2 -10105.916} C_VEL
LIN {X 0,Y 418.219,Z 306.326,A -85,B 0,C 180,E1 -10109.166,E2 -10109.166} C_VEL
LIN {X 0,Y 418.326,Z 300.709,A -85,B 0,C 180,E1 -10111.952,E2 -10111.952} C_VEL
LIN {X 0,Y 418.133,Z 297.404,A -85,B 0,C 180,E1 -10113.569,E2 -10113.569} C_VEL
LIN {X 0,Y 418.239,Z 297.391,A -85,B 0,C 180,E1 -10116.236,E2 -10116.236} C_VEL
LIN {X 0,Y 418.246,Z 297.387,A -85,B 0,C 180,E1 -10119.683,E2 -10119.683} C_VEL
LIN {X 0,Y 418.226,Z 297.39,A -85,B 0,C 180,E1 -10122.32,E2 -10122.32} C_VEL
LIN {X 0,Y 418.25,Z 297.532,A -85,B 0,C 180,E1 -10125.953,E2 -10125.953} C_VEL
LIN {X 0,Y 419.768,Z 305.099,A -85,B 0,C 180,E1 -10129.235,E2 -10129.235} C_VEL
LIN {X 0,Y 420.965,Z 311.418,A -85,B 0,C 180,E1 -10131.85,E2 -10131.85} C_VEL
LIN {X 0,Y 421.501,Z 316.202,A -85,B 0,C 180,E1 -10133.74,E2 -10133.74} C_VEL
LIN {X 0,Y 420.827,Z 324.013,A -85,B 0,C 180,E1 -10136.618,E2 -10136.618} C_VEL
LIN {X 0,Y 420.173,Z 333.121,A -85,B 0,C 180,E1 -10139.881,E2 -10139.881} C_VEL
LIN {X 0,Y 419.485,Z 342.37,A -85,B 0,C 180,E1 -10143.105,E2 -10143.105} C_VEL
LIN {X 0,Y 418.953,Z 351.634,A -85,B 0,C 180,E1 -10146.259,E2 -10146.259} C_VEL
LIN {X 0,Y 418.392,Z 362.326,A -85,B 0,C 180,E1 -10149.826,E2 -10149.826} C_VEL
LIN {X 0,Y 417.995,Z 370.932,A -85,B 0,C 180,E1 -10152.645,E2 -10152.645} C_VEL
LIN {X 0,Y 420.227,Z 386.343,A -85,B 0,C 180,E1 -10153.24,E2 -10153.24} C_VEL
LIN {X 0,Y 421.809,Z 398.032,A -85,B 0,C 180,E1 -10153.857,E2 -10153.857} C_VEL
LIN {X 0,Y 421.104,Z 410.633,A -85,B 0,C 180,E1 -10154.636,E2 -10154.636} C_VEL
LIN {X 0,Y 420.27,Z 422.603,A -85,B 0,C 180,E1 -10155.595,E2 -10155.595} C_VEL
LIN {X 0,Y 419.607,Z 433.308,A -85,B 0,C 180,E1 -10156.685,E2 -10156.685} C_VEL
LIN {X 0,Y 418.94,Z 442.979,A -85,B 0,C 180,E1 -10157.895,E2 -10157.895} C_VEL
LIN {X 0,Y 418.333,Z 450.941,A -85,B 0,C 180,E1 -10159.106,E2 -10159.106} C_VEL
LIN {X 0,Y 417.851,Z 458.769,A -85,B 0,C 180,E1 -10160.561,E2 -10160.561} C_VEL
LIN {X 0,Y 417.542,Z 464.106,A -85,B 0,C 180,E1 -10161.774,E2 -10161.774} C_VEL
LIN {X 0,Y 417.296,Z 470.258,A -85,B 0,C 180,E1 -10163.548,E2 -10163.548} C_VEL
LIN {X 0,Y 417.168,Z 474.418,A -85,B 0,C 180,E1 -10165.168,E2 -10165.168} C_VEL
LIN {X 0,Y 417.075,Z 476.3,A -85,B 0,C 180,E1 -10166.135,E2 -10166.135} C_VEL
LIN {X 0,Y 417.149,Z 477.726,A -85,B 0,C 180,E1 -10167.103,E2 -10167.103} C_VEL
LIN {X 0,Y 417.15,Z 479.314,A -85,B 0,C 180,E1 -10169.035,E2 -10169.035} C_VEL
LIN {X 0,Y 417.122,Z 479.505,A -85,B 0,C 180,E1 -10170,E2 -10170} C_VEL
LIN {X 0,Y 417.151,Z 479.258,A -85,B 0,C 180,E1 -10170.965,E2 -10170.965} C_VEL
LIN {X 0,Y 417.135,Z 478.592,A -85,B 0,C 180,E1 -10171.931,E2 -10171.931} C_VEL
LIN {X 0,Y 417.152,Z 477.526,A -85,B 0,C 180,E1 -10172.897,E2 -10172.897} C_VEL
LIN {X 0,Y 417.095,Z 476.037,A -85,B 0,C 180,E1 -10173.865,E2 -10173.865} C_VEL
LIN {X 0,Y 417.259,Z 472.958,A -85,B 0,C 180,E1 -10175.315,E2 -10175.315} C_VEL
LIN {X 0,Y 417.32,Z 468.791,A -85,B 0,C 180,E1 -10176.77,E2 -10176.77} C_VEL
LIN {X 0,Y 417.629,Z 462.414,A -85,B 0,C 180,E1 -10178.468,E2 -10178.468} C_VEL
LIN {X 0,Y 417.991,Z 455.478,A -85,B 0,C 180,E1 -10179.924,E2 -10179.924} C_VEL
LIN {X 0,Y 418.527,Z 446.916,A -85,B 0,C 180,E1 -10181.38,E2 -10181.38} C_VEL
LIN {X 0,Y 419.092,Z 438.146,A -85,B 0,C 180,E1 -10182.592,E2 -10182.592} C_VEL
LIN {X 0,Y 419.747,Z 429.004,A -85,B 0,C 180,E1 -10183.639,E2 -10183.639} C_VEL
LIN {X 0,Y 420.415,Z 416.918,A -85,B 0,C 180,E1 -10184.77,E2 -10184.77} C_VEL
LIN {X 0,Y 421.244,Z 405.576,A -85,B 0,C 180,E1 -10185.607,E2 -10185.607} C_VEL
LIN {X 0,Y 421.535,Z 396.445,A -85,B 0,C 180,E1 -10186.154,E2 -10186.154} C_VEL
LIN {X 0,Y 419.786,Z 383.217,A -85,B 0,C 180,E1 -10186.854,E2 -10186.854} C_VEL
LIN {X 0,Y 417.95,Z 368.485,A -85,B 0,C 180,E1 -10187.446,E2 -10187.446} C_VEL
LIN {X 0,Y 418.262,Z 358.341,A -85,B 0,C 180,E1 -10190.662,E2 -10190.662} C_VEL
LIN {X 0,Y 418.71,Z 348.807,A -85,B 0,C 180,E1 -10193.756,E2 -10193.756} C_VEL
LIN {X 0,Y 419.179,Z 339.395,A -85,B 0,C 180,E1 -10196.916,E2 -10196.916} C_VEL
LIN {X 0,Y 419.758,Z 330.22,A -85,B 0,C 180,E1 -10200.152,E2 -10200.152} C_VEL
LIN {X 0,Y 420.48,Z 321.43,A -85,B 0,C 180,E1 -10203.475,E2 -10203.475} C_VEL
LIN {X 0,Y 421.192,Z 314.721,A -85,B 0,C 180,E1 -10206.253,E2 -10206.253} C_VEL
LIN {X 0,Y 420.753,Z 310.555,A -85,B 0,C 180,E1 -10208.274,E2 -10208.274} C_VEL
LIN {X 0,Y 419.875,Z 305.551,A -85,B 0,C 180,E1 -10211.129,E2 -10211.129} C_VEL
LIN {X 0,Y 419.125,Z 301.787,A -85,B 0,C 180,E1 -10213.86,E2 -10213.86} C_VEL
LIN {X 0,Y 418.598,Z 299.121,A -85,B 0,C 180,E1 -10216.499,E2 -10216.499} C_VEL
LIN {X 0,Y 418.223,Z 297.421,A -85,B 0,C 180,E1 -10219.131,E2 -10219.131} C_VEL
LIN {X 0,Y 418.228,Z 297.391,A -85,B 0,C 180,E1 -10222.167,E2 -10222.167} C_VEL
LIN {X 0,Y 418.268,Z 297.387,A -85,B 0,C 180,E1 -10225.42,E2 -10225.42} C_VEL
LIN {X 0,Y 418.215,Z 297.402,A -85,B 0,C 180,E1 -10228.604,E2 -10228.604} C_VEL
LIN {X 0,Y 418.518,Z 298.853,A -85,B 0,C 180,E1 -10231.953,E2 -10231.953} C_VEL
LIN {X 0,Y 418.714,Z 300.675,A -85,B 0,C 180,E1 -10235.189,E2 -10235.189} C_VEL
LIN {X 0,Y 418.652,Z 302.751,A -85,B 0,C 180,E1 -10238.326,E2 -10238.326} C_VEL
LIN {X 0,Y 418.491,Z 304.99,A -85,B 0,C 180,E1 -10241.393,E2 -10241.393} C_VEL
LIN {X 0,Y 418.436,Z 306.125,A -85,B 0,C 180,E1 -10242.841,E2 -10242.841} C_VEL
LIN {X 0,Y 422.518,Z 318.307,A -85,B 0,C 180,E1 -10243.574,E2 -10243.574} C_VEL
LIN {X 0,Y 422.949,Z 320.765,A -85,B 0,C 180,E1 -10243.716,E2 -10243.716} C_VEL
LIN {X 0,Y 422.467,Z 333.39,A -85,B 0,C 180,E1 -10244.44,E2 -10244.44} C_VEL
LIN {X 0,Y 421.813,Z 345.967,A -85,B 0,C 180,E1 -10245.38,E2 -10245.38} C_VEL
LIN {X 0,Y 421.061,Z 357.471,A -85,B 0,C 180,E1 -10246.486,E2 -10246.486} C_VEL
LIN {X 0,Y 420.426,Z 367.53,A -85,B 0,C 180,E1 -10247.694,E2 -10247.694} C_VEL
LIN {X 0,Y 419.844,Z 375.724,A -85,B 0,C 180,E1 -10248.901,E2 -10248.901} C_VEL
LIN {X 0,Y 419.168,Z 383.726,A -85,B 0,C 180,E1 -10250.348,E2 -10250.348} C_VEL
LIN {X 0,Y 418.771,Z 390.298,A -85,B 0,C 180,E1 -10251.847,E2 -10251.847} C_VEL
LIN {X 0,Y 418.237,Z 395.153,A -85,B 0,C 180,E1 -10253.245,E2 -10253.245} C_VEL
LIN {X 0,Y 418.063,Z 398.976,A -85,B 0,C 180,E1 -10254.695,E2 -10254.695} C_VEL
LIN {X 0,Y 417.799,Z 401.754,A -85,B 0,C 180,E1 -10256.142,E2 -10256.142} C_VEL
LIN {X 0,Y 417.55,Z 403.045,A -85,B 0,C 180,E1 -10257.106,E2 -10257.106} C_VEL
LIN {X 0,Y 417.399,Z 403.915,A -85,B 0,C 180,E1 -10258.07,E2 -10258.07} C_VEL
LIN {X 0,Y 417.336,Z 404.377,A -85,B 0,C 180,E1 -10259.035,E2 -10259.035} C_VEL
LIN {X 0,Y 417.304,Z 404.404,A -85,B 0,C 180,E1 -10260,E2 -10260} C_VEL
LIN {X 0,Y 417.303,Z 404.001,A -85,B 0,C 180,E1 -10260.965,E2 -10260.965} C_VEL
LIN {X 0,Y 417.368,Z 403.191,A -85,B 0,C 180,E1 -10261.93,E2 -10261.93} C_VEL
LIN {X 0,Y 417.537,Z 401.967,A -85,B 0,C 180,E1 -10262.895,E2 -10262.895} C_VEL
LIN {X 0,Y 417.799,Z 399.295,A -85,B 0,C 180,E1 -10264.341,E2 -10264.341} C_VEL
LIN {X 0,Y 417.816,Z 395.61,A -85,B 0,C 180,E1 -10265.792,E2 -10265.792} C_VEL
LIN {X 0,Y 418.094,Z 390.332,A -85,B 0,C 180,E1 -10267.355,E2 -10267.355} C_VEL
LIN {X 0,Y 418.477,Z 383.472,A -85,B 0,C 180,E1 -10268.937,E2 -10268.937} C_VEL
LIN {X 0,Y 418.937,Z 375.583,A -85,B 0,C 180,E1 -10270.39,E2 -10270.39} C_VEL
LIN {X 0,Y 419.423,Z 367.506,A -85,B 0,C 180,E1 -10271.6,E2 -10271.6} C_VEL
LIN {X 0,Y 420.03,Z 356.602,A -85,B 0,C 180,E1 -10272.932,E2 -10272.932} C_VEL
LIN {X 0,Y 420.592,Z 345.982,A -85,B 0,C 180,E1 -10273.977,E2 -10273.977} C_VEL
LIN {X 0,Y 421.02,Z 334.678,A -85,B 0,C 180,E1 -10274.872,E2 -10274.872} C_VEL
LIN {X 0,Y 421.601,Z 321.703,A -85,B 0,C 180,E1 -10275.67,E2 -10275.67} C_VEL
LIN {X 0,Y 421.502,Z 316.274,A -85,B 0,C 180,E1 -10275.948,E2 -10275.948} C_VEL
LIN {X 0,Y 418.27,Z 302.709,A -85,B 0,C 180,E1 -10276.587,E2 -10276.587} C_VEL
LIN {X 0,Y 417.583,Z 299.681,A -85,B 0,C 180,E1 -10276.727,E2 -10276.727} C_VEL
LIN {X 0,Y 417.551,Z 297.477,A -85,B 0,C 180,E1 -10278.651,E2 -10278.651} C_VEL
LIN {X 0,Y 417.889,Z 297.428,A -85,B 0,C 180,E1 -10281.715,E2 -10281.715} C_VEL
LIN {X 0,Y 418.195,Z 297.392,A -85,B 0,C 180,E1 -10284.844,E2 -10284.844} C_VEL
LIN {X 0,Y 418.286,Z 297.378,A -85,B 0,C 180,E1 -10288.064,E2 -10288.064} C_VEL
LIN {X 0,Y 418.214,Z 297.383,A -85,B 0,C 180,E1 -10291.396,E2 -10291.396} C_VEL
LIN {X 0,Y 418.268,Z 297.381,A -85,B 0,C 180,E1 -10294.58,E2 -10294.58} C_VEL
LIN {X 0,Y 418.231,Z 297.391,A -85,B 0,C 180,E1 -10297.833,E2 -10297.833} C_VEL
LIN {X 0,Y 418.225,Z 297.389,A -85,B 0,C 180,E1 -10300.948,E2 -10300.948} C_VEL
LIN {X 0,Y 418.215,Z 297.394,A -85,B 0,C 180,E1 -10303.73,E2 -10303.73} C_VEL
LIN {X 0,Y 418.212,Z 297.388,A -85,B 0,C 180,E1 -10306.449,E2 -10306.449} C_VEL
LIN {X 0,Y 418.225,Z 297.388,A -85,B 0,C 180,E1 -10309.13,E2 -10309.13} C_VEL
